C07307=1196.798,-117.716,-38.515,179.057,5.551,149.259
C07308=1196.792,-117.467,-38.525,179.060,5.552,149.258
C07309=1196.787,-117.217,-38.534,179.061,5.552,149.258
C07310=1196.782,-116.967,-38.543,179.064,5.552,149.257
C07311=1196.777,-116.718,-38.553,179.066,5.552,149.256
C07312=1196.771,-116.468,-38.562,179.068,5.553,149.256
C07313=1196.766,-116.219,-38.572,179.070,5.552,149.255
C07314=1196.761,-115.968,-38.581,179.072,5.553,149.255
C07315=1196.755,-115.718,-38.590,179.075,5.553,149.254
C07316=1196.750,-115.469,-38.600,179.077,5.553,149.253
C07317=1196.745,-115.219,-38.609,179.079,5.553,149.253
C07318=1196.739,-114.969,-38.618,179.081,5.553,149.252
C07319=1196.734,-114.719,-38.629,179.084,5.553,149.251
C07320=1196.729,-114.469,-38.637,179.086,5.554,149.251
C07321=1196.724,-114.220,-38.648,179.088,5.553,149.250
C07322=1196.719,-113.970,-38.657,179.090,5.554,149.250
C07323=1196.714,-113.721,-38.666,179.092,5.554,149.249
C07324=1196.708,-113.470,-38.676,179.095,5.554,149.248
C07325=1196.703,-113.221,-38.685,179.096,5.554,149.248
C07326=1196.697,-112.971,-38.695,179.099,5.555,149.247
C07327=1196.692,-112.721,-38.704,179.101,5.554,149.246
C07328=1196.686,-112.472,-38.714,179.103,5.555,149.246
C07329=1196.681,-112.222,-38.723,179.105,5.555,149.245
C07330=1196.675,-111.972,-38.733,179.108,5.555,149.245
C07331=1196.670,-111.722,-38.742,179.110,5.555,149.244
C07332=1196.666,-111.472,-38.752,179.112,5.555,149.243
C07333=1196.660,-111.222,-38.761,179.114,5.555,149.243
C07334=1196.655,-110.973,-38.771,179.117,5.556,149.242
C07335=1196.649,-110.723,-38.780,179.119,5.555,149.241
C07336=1196.645,-110.474,-38.790,179.121,5.556,149.241
C07337=1196.639,-110.223,-38.800,179.123,5.556,149.240
C07338=1196.634,-109.974,-38.809,179.125,5.557,149.240
C07339=1196.628,-109.724,-38.819,179.127,5.556,149.239
C07340=1196.624,-109.474,-38.829,179.130,5.557,149.238
C07341=1196.618,-109.224,-38.838,179.132,5.557,149.238
C07342=1196.613,-108.975,-38.848,179.134,5.557,149.237
C07343=1196.607,-108.725,-38.858,179.136,5.557,149.236
C07344=1196.602,-108.475,-38.867,179.139,5.557,149.236
C07345=1196.596,-108.226,-38.877,179.141,5.557,149.235
C07346=1196.591,-107.976,-38.886,179.143,5.557,149.234
C07347=1196.586,-107.726,-38.897,179.145,5.557,149.234
C07348=1196.581,-107.476,-38.906,179.148,5.558,149.233
C07349=1196.576,-107.226,-38.916,179.149,5.558,149.233
C07350=1196.570,-106.977,-38.926,179.152,5.558,149.232
C07351=1196.565,-106.727,-38.935,179.154,5.558,149.231
C07352=1196.559,-106.477,-38.945,179.156,5.559,149.231
C07353=1196.554,-106.228,-38.955,179.158,5.558,149.230
C07354=1196.549,-105.977,-38.964,179.161,5.559,149.229
C07355=1196.544,-105.728,-38.974,179.163,5.559,149.229
C07356=1196.539,-105.478,-38.984,179.165,5.559,149.228
C07357=1196.533,-105.229,-38.993,179.167,5.559,149.227
C07358=1196.528,-104.979,-39.003,179.169,5.559,149.227
C07359=1196.523,-104.729,-39.014,179.172,5.559,149.226
C07360=1196.518,-104.479,-39.023,179.174,5.559,149.225
C07361=1196.512,-104.229,-39.033,179.176,5.560,149.225
C07362=1196.507,-103.980,-39.043,179.178,5.560,149.224
C07363=1196.501,-103.730,-39.052,179.181,5.560,149.224
C07364=1196.496,-103.480,-39.063,179.183,5.560,149.223
C07365=1196.491,-103.231,-39.072,179.185,5.561,149.222
C07366=1196.486,-102.980,-39.082,179.188,5.560,149.222
C07367=1196.481,-102.731,-39.091,179.190,5.561,149.221
C07368=1196.476,-102.481,-39.102,179.192,5.561,149.220
C07369=1196.470,-102.231,-39.112,179.194,5.561,149.220
C07370=1196.465,-101.982,-39.121,179.196,5.561,149.219
C07371=1196.459,-101.710,-39.133,179.199,5.561,149.219
C07372=1196.453,-101.439,-39.143,179.201,5.562,149.218
C07373=1196.448,-101.167,-39.153,179.204,5.561,149.217
C07374=1196.442,-100.896,-39.165,179.206,5.562,149.216
C07375=1196.437,-100.647,-39.175,179.208,5.562,149.216
C07376=1196.431,-100.396,-39.184,179.210,5.562,149.215
C07377=1196.426,-100.146,-39.195,179.213,5.562,149.215
C07378=1196.421,-99.897,-39.204,179.215,5.562,149.214
C07379=1196.416,-99.647,-39.214,179.217,5.563,149.213
C07380=1196.410,-99.398,-39.225,179.220,5.563,149.213
C07381=1196.406,-99.148,-39.235,179.222,5.563,149.212
C07382=1196.400,-98.898,-39.244,179.224,5.563,149.211
C07383=1196.394,-98.648,-39.254,179.226,5.563,149.211
C07384=1196.389,-98.398,-39.265,179.229,5.563,149.210
C07385=1196.384,-98.149,-39.275,179.231,5.564,149.209
C07386=1196.379,-97.899,-39.285,179.233,5.563,149.209
C07387=1196.373,-97.650,-39.295,179.236,5.564,149.208
C07388=1196.369,-97.399,-39.304,179.237,5.564,149.208
C07389=1196.363,-97.150,-39.314,179.240,5.564,149.207
C07390=1196.357,-96.900,-39.325,179.242,5.564,149.206
C07391=1196.352,-96.650,-39.335,179.244,5.565,149.206
C07392=1196.347,-96.401,-39.345,179.246,5.564,149.205
C07393=1196.342,-96.151,-39.355,179.249,5.565,149.204
C07394=1196.336,-95.901,-39.365,179.251,5.565,149.204
C07395=1196.331,-95.651,-39.376,179.253,5.565,149.203
C07396=1196.326,-95.402,-39.386,179.256,5.565,149.202
C07397=1196.321,-95.152,-39.396,179.257,5.565,149.202
C07398=1196.316,-94.902,-39.406,179.260,5.566,149.201
C07399=1196.310,-94.652,-39.416,179.262,5.566,149.200
C07400=1196.304,-94.402,-39.426,179.265,5.566,149.200
C07401=1196.300,-94.153,-39.436,179.266,5.566,149.199
C07402=1196.294,-93.903,-39.446,179.269,5.566,149.199
C07403=1196.289,-93.653,-39.456,179.271,5.566,149.198
C07404=1196.284,-93.403,-39.467,179.273,5.567,149.197
C07405=1196.278,-93.154,-39.477,179.276,5.567,149.197
C07406=1196.273,-92.904,-39.487,179.278,5.567,149.196
C07407=1196.268,-92.654,-39.497,179.280,5.568,149.195
C07408=1196.263,-92.405,-39.508,179.282,5.567,149.195
C07409=1196.257,-92.155,-39.518,179.285,5.568,149.194
C07410=1196.252,-91.905,-39.528,179.287,5.568,149.194
C07411=1196.247,-91.655,-39.539,179.289,5.568,149.193
C07412=1196.241,-91.406,-39.549,179.291,5.568,149.192
C07413=1196.237,-91.156,-39.559,179.294,5.568,149.191
C07414=1196.231,-90.906,-39.569,179.296,5.569,149.191
C07415=1196.226,-90.656,-39.579,179.298,5.568,149.190
C07416=1196.221,-90.406,-39.590,179.301,5.569,149.189
C07417=1196.215,-90.158,-39.601,179.303,5.569,149.189
C07418=1196.210,-89.907,-39.611,179.305,5.569,149.188
C07419=1196.205,-89.658,-39.621,179.307,5.569,149.188
C07420=1196.200,-89.408,-39.631,179.310,5.569,149.187
C07421=1196.195,-89.158,-39.642,179.312,5.569,149.186
C07422=1196.189,-88.909,-39.652,179.314,5.570,149.186
C07423=1196.184,-88.659,-39.662,179.317,5.570,149.185
C07424=1196.179,-88.409,-39.673,179.319,5.570,149.184
C07425=1196.174,-88.159,-39.683,179.321,5.571,149.184
C07426=1196.168,-87.909,-39.693,179.323,5.570,149.183
C07427=1196.163,-87.660,-39.704,179.326,5.571,149.183
C07428=1196.158,-87.410,-39.715,179.328,5.571,149.182
C07429=1196.152,-87.160,-39.725,179.330,5.571,149.181
C07430=1196.147,-86.910,-39.736,179.333,5.571,149.180
C07431=1196.142,-86.661,-39.745,179.335,5.571,149.180
C07432=1196.137,-86.411,-39.756,179.337,5.572,149.179
C07433=1196.132,-86.162,-39.767,179.339,5.571,149.179
C07434=1196.126,-85.912,-39.777,179.342,5.572,149.178
C07435=1196.121,-85.662,-39.788,179.344,5.572,149.177
C07436=1196.116,-85.413,-39.798,179.346,5.572,149.177
C07437=1196.111,-85.162,-39.808,179.349,5.573,149.176
C07438=1196.106,-84.913,-39.819,179.351,5.573,149.175
C07439=1196.101,-84.663,-39.830,179.353,5.573,149.175
C07440=1196.095,-84.414,-39.840,179.355,5.573,149.174
C07441=1196.090,-84.163,-39.851,179.358,5.573,149.173
C07442=1196.084,-83.914,-39.861,179.360,5.573,149.173
C07443=1196.080,-83.664,-39.872,179.362,5.574,149.172
C07444=1196.074,-83.415,-39.882,179.365,5.574,149.171
C07445=1196.069,-83.164,-39.893,179.367,5.574,149.171
C07446=1196.063,-82.915,-39.903,179.369,5.574,149.170
C07447=1196.059,-82.665,-39.914,179.371,5.574,149.170
C07448=1196.053,-82.416,-39.925,179.374,5.575,149.169
C07449=1196.048,-82.166,-39.935,179.376,5.575,149.168
C07450=1196.043,-81.916,-39.946,179.378,5.575,149.168
C07451=1196.037,-81.667,-39.956,179.381,5.575,149.167
C07452=1196.032,-81.417,-39.967,179.383,5.575,149.166
C07453=1196.027,-81.167,-39.977,179.385,5.576,149.166
C07454=1196.022,-80.918,-39.988,179.387,5.575,149.165
C07455=1196.016,-80.668,-39.999,179.390,5.576,149.164
C07456=1196.011,-80.418,-40.009,179.392,5.577,149.164
C07457=1196.006,-80.168,-40.021,179.394,5.576,149.163
C07458=1196.000,-79.918,-40.031,179.397,5.577,149.162
C07459=1195.996,-79.669,-40.043,179.399,5.576,149.162
C07460=1195.990,-79.419,-40.053,179.401,5.577,149.161
C07461=1195.985,-79.169,-40.063,179.404,5.578,149.161
C07462=1195.980,-78.920,-40.074,179.406,5.577,149.160
C07463=1195.975,-78.670,-40.085,179.409,5.578,149.159
C07464=1195.969,-78.420,-40.095,179.410,5.578,149.159
C07465=1195.964,-78.170,-40.106,179.413,5.578,149.158
C07466=1195.959,-77.921,-40.117,179.415,5.578,149.157
C07467=1195.953,-77.671,-40.128,179.418,5.578,149.156
C07468=1195.948,-77.421,-40.139,179.420,5.579,149.156
C07469=1195.943,-77.171,-40.149,179.422,5.578,149.155
C07470=1195.938,-76.922,-40.160,179.425,5.579,149.155
C07471=1195.933,-76.672,-40.171,179.426,5.579,149.154
C07472=1195.928,-76.422,-40.182,179.429,5.579,149.153
C07473=1195.922,-76.173,-40.192,179.431,5.580,149.153
C07474=1195.917,-75.923,-40.204,179.434,5.579,149.152
C07475=1195.911,-75.652,-40.215,179.436,5.580,149.151
C07476=1195.905,-75.381,-40.227,179.439,5.580,149.151
C07477=1195.900,-75.110,-40.239,179.442,5.581,149.150
C07478=1195.894,-74.840,-40.250,179.444,5.580,149.149
C07479=1195.889,-74.590,-40.262,179.446,5.581,149.149
C07480=1195.884,-74.340,-40.273,179.448,5.581,149.148
C07481=1195.878,-74.091,-40.283,179.451,5.581,149.147
C07482=1195.874,-73.841,-40.294,179.453,5.582,149.147
C07483=1195.868,-73.592,-40.305,179.455,5.582,149.146
C07484=1195.863,-73.342,-40.316,179.458,5.582,149.145
C07485=1195.858,-73.091,-40.327,179.460,5.582,149.145
C07486=1195.852,-72.842,-40.338,179.462,5.582,149.144
C07487=1195.847,-72.592,-40.349,179.464,5.583,149.143
C07488=1195.841,-72.343,-40.360,179.467,5.583,149.143
C07489=1195.837,-72.093,-40.371,179.469,5.583,149.142
C07490=1195.832,-71.843,-40.382,179.472,5.583,149.141
C07491=1195.826,-71.594,-40.393,179.473,5.583,149.141
C07492=1195.821,-71.344,-40.404,179.476,5.584,149.140
C07493=1195.815,-71.095,-40.415,179.478,5.583,149.139
C07494=1195.810,-70.844,-40.426,179.481,5.584,149.139
C07495=1195.806,-70.595,-40.437,179.483,5.585,149.138
C07496=1195.800,-70.346,-40.448,179.485,5.584,149.138
C07497=1195.795,-70.095,-40.459,179.488,5.585,149.137
C07498=1195.790,-69.846,-40.470,179.491,5.585,149.136
C07499=1195.785,-69.597,-40.481,179.492,5.585,149.136
C07500=1195.779,-69.346,-40.492,179.495,5.586,149.135
C07501=1195.774,-69.097,-40.504,179.497,5.585,149.134
C07502=1195.769,-68.848,-40.515,179.500,5.586,149.134
C07503=1195.763,-68.597,-40.526,179.502,5.586,149.133
C07504=1195.758,-68.347,-40.537,179.504,5.586,149.132
C07505=1195.753,-68.099,-40.548,179.506,5.587,149.132
C07506=1195.747,-67.848,-40.559,179.509,5.587,149.131
C07507=1195.743,-67.598,-40.570,179.511,5.587,149.130
C07508=1195.737,-67.349,-40.581,179.513,5.587,149.130
C07509=1195.732,-67.099,-40.592,179.515,5.587,149.129
C07510=1195.727,-66.849,-40.604,179.518,5.587,149.128
C07511=1195.722,-66.600,-40.615,179.521,5.588,149.128
C07512=1195.716,-66.350,-40.627,179.522,5.588,149.127
C07513=1195.711,-66.100,-40.637,179.525,5.588,149.126
C07514=1195.707,-65.851,-40.648,179.528,5.589,149.126
C07515=1195.701,-65.601,-40.660,179.530,5.588,149.125
C07516=1195.696,-65.352,-40.671,179.532,5.589,149.125
C07517=1195.691,-65.101,-40.682,179.535,5.590,149.124
C07518=1195.685,-64.851,-40.694,179.537,5.589,149.123
C07519=1195.680,-64.603,-40.705,179.539,5.590,149.122
C07520=1195.675,-64.353,-40.717,179.541,5.590,149.122
C07521=1195.670,-64.102,-40.727,179.544,5.590,149.121
C07522=1195.664,-63.853,-40.738,179.546,5.591,149.121
C07523=1195.659,-63.604,-40.750,179.548,5.590,149.120
C07524=1195.654,-63.354,-40.761,179.551,5.591,149.119
C07525=1195.649,-63.104,-40.773,179.553,5.592,149.119
C07526=1195.644,-62.855,-40.784,179.555,5.591,149.118
C07527=1195.639,-62.605,-40.795,179.558,5.592,149.117
C07528=1195.633,-62.355,-40.806,179.561,5.592,149.117
C07529=1195.628,-62.105,-40.818,179.562,5.592,149.116
C07530=1195.623,-61.855,-40.830,179.565,5.592,149.115
C07531=1195.618,-61.606,-40.841,179.568,5.593,149.115
C07532=1195.612,-61.356,-40.852,179.570,5.593,149.114
C07533=1195.608,-61.107,-40.864,179.572,5.593,149.113
C07534=1195.602,-60.856,-40.875,179.575,5.594,149.113
C07535=1195.597,-60.607,-40.886,179.577,5.593,149.112
C07536=1195.591,-60.357,-40.898,179.579,5.594,149.111
C07537=1195.586,-60.108,-40.909,179.582,5.594,149.111
C07538=1195.582,-59.858,-40.920,179.584,5.594,149.110
C07539=1195.576,-59.608,-40.932,179.586,5.595,149.109
C07540=1195.571,-59.359,-40.943,179.588,5.594,149.109
C07541=1195.566,-59.109,-40.955,179.591,5.595,149.108
C07542=1195.561,-58.860,-40.966,179.593,5.596,149.108
C07543=1195.556,-58.610,-40.978,179.595,5.595,149.107
C07544=1195.551,-58.360,-40.989,179.598,5.596,149.106
C07545=1195.545,-58.110,-41.001,179.601,5.596,149.105
C07546=1195.540,-57.861,-41.012,179.603,5.596,149.105
C07547=1195.535,-57.611,-41.024,179.605,5.597,149.104
C07548=1195.529,-57.361,-41.036,179.608,5.597,149.104
C07549=1195.525,-57.112,-41.047,179.610,5.597,149.103
C07550=1195.519,-56.862,-41.059,179.612,5.597,149.102
C07551=1195.514,-56.612,-41.070,179.614,5.598,149.102
C07552=1195.508,-56.363,-41.082,179.617,5.598,149.101
C07553=1195.504,-56.113,-41.093,179.619,5.598,149.100
C07554=1195.498,-55.863,-41.105,179.622,5.598,149.100
C07555=1195.494,-55.614,-41.116,179.624,5.598,149.099
C07556=1195.488,-55.364,-41.128,179.626,5.599,149.098
C07557=1195.483,-55.114,-41.140,179.629,5.599,149.098
C07558=1195.478,-54.864,-41.152,179.631,5.599,149.097
C07559=1195.472,-54.615,-41.163,179.634,5.599,149.096
C07560=1195.467,-54.365,-41.174,179.636,5.600,149.096
C07561=1195.462,-54.116,-41.186,179.638,5.601,149.095
C07562=1195.457,-53.866,-41.198,179.640,5.600,149.094
C07563=1195.452,-53.616,-41.209,179.643,5.601,149.094
C07564=1195.447,-53.367,-41.222,179.646,5.601,149.093
C07565=1195.442,-53.117,-41.233,179.647,5.601,149.093
C07566=1195.437,-52.867,-41.245,179.650,5.602,149.092
C07567=1195.431,-52.617,-41.257,179.653,5.602,149.091
C07568=1195.426,-52.368,-41.268,179.655,5.602,149.090
C07569=1195.420,-52.118,-41.280,179.657,5.602,149.090
C07570=1195.416,-51.869,-41.291,179.660,5.603,149.089
C07571=1195.410,-51.619,-41.303,179.662,5.603,149.089
C07572=1195.405,-51.369,-41.316,179.664,5.603,149.088
C07573=1195.400,-51.120,-41.327,179.667,5.604,149.087
C07574=1195.395,-50.870,-41.339,179.669,5.604,149.087
C07575=1195.390,-50.620,-41.351,179.671,5.604,149.086
C07576=1195.385,-50.370,-41.362,179.674,5.604,149.085
C07577=1195.380,-50.121,-41.375,179.677,5.605,149.085
C07578=1195.374,-49.871,-41.386,179.679,5.605,149.084
C07579=1195.368,-49.601,-41.399,179.681,5.605,149.083
C07580=1195.363,-49.331,-41.412,179.684,5.605,149.082
C07581=1195.358,-49.061,-41.425,179.687,5.606,149.082
C07582=1195.352,-48.791,-41.438,179.689,5.606,149.081
C07583=1195.346,-48.541,-41.450,179.691,5.606,149.081
C07584=1195.341,-48.291,-41.461,179.694,5.607,149.080
C07585=1195.336,-48.042,-41.473,179.696,5.607,149.079
C07586=1195.331,-47.792,-41.485,179.698,5.607,149.078
C07587=1195.326,-47.542,-41.497,179.701,5.607,149.078
C07588=1195.320,-47.292,-41.509,179.703,5.608,149.077
C07589=1195.316,-47.043,-41.520,179.705,5.608,149.077
C07590=1195.311,-46.793,-41.533,179.708,5.608,149.076
C07591=1195.305,-46.543,-41.545,179.711,5.609,149.075
C07592=1195.300,-46.294,-41.557,179.713,5.609,149.074
C07593=1195.295,-46.045,-41.569,179.715,5.609,149.074
C07594=1195.290,-45.795,-41.581,179.718,5.610,149.073
C07595=1195.284,-45.545,-41.592,179.720,5.610,149.073
C07596=1195.279,-45.295,-41.605,179.722,5.610,149.072
C07597=1195.274,-45.045,-41.617,179.725,5.610,149.071
C07598=1195.269,-44.796,-41.628,179.727,5.611,149.071
C07599=1195.264,-44.546,-41.641,179.730,5.611,149.070
C07600=1195.259,-44.296,-41.653,179.732,5.611,149.069
C07601=1195.253,-44.047,-41.665,179.735,5.612,149.069
C07602=1195.248,-43.797,-41.677,179.737,5.612,149.068
C07603=1195.243,-43.548,-41.689,179.739,5.612,149.067
C07604=1195.238,-43.298,-41.701,179.742,5.612,149.067
C07605=1195.233,-43.048,-41.713,179.744,5.613,149.066
C07606=1195.227,-42.798,-41.725,179.747,5.613,149.065
C07607=1195.222,-42.549,-41.737,179.749,5.613,149.065
C07608=1195.217,-42.299,-41.749,179.751,5.614,149.064
C07609=1195.212,-42.050,-41.761,179.754,5.614,149.063
C07610=1195.207,-41.800,-41.773,179.756,5.614,149.063
C07611=1195.202,-41.551,-41.786,179.759,5.614,149.062
C07612=1195.196,-41.301,-41.798,179.761,5.615,149.062
C07613=1195.191,-41.052,-41.810,179.763,5.616,149.061
C07614=1195.186,-40.802,-41.822,179.765,5.615,149.060
C07615=1195.181,-40.552,-41.835,179.768,5.616,149.059
C07616=1195.176,-40.302,-41.847,179.771,5.616,149.059
C07617=1195.171,-40.052,-41.860,179.773,5.617,149.058
C07618=1195.166,-39.803,-41.871,179.775,5.617,149.058
C07619=1195.161,-39.554,-41.884,179.778,5.617,149.057
C07620=1195.156,-39.304,-41.895,179.780,5.618,149.056
C07621=1195.150,-39.054,-41.908,179.783,5.618,149.056
C07622=1195.145,-38.804,-41.920,179.785,5.618,149.055
C07623=1195.140,-38.555,-41.933,179.787,5.619,149.054
C07624=1195.134,-38.305,-41.944,179.790,5.619,149.054
C07625=1195.129,-38.056,-41.957,179.792,5.619,149.053
C07626=1195.124,-37.806,-41.969,179.795,5.619,149.052
C07627=1195.119,-37.556,-41.982,179.797,5.620,149.052
C07628=1195.114,-37.306,-41.994,179.800,5.620,149.051
C07629=1195.109,-37.057,-42.006,179.802,5.620,149.050
C07630=1195.104,-36.807,-42.019,179.804,5.621,149.050
C07631=1195.098,-36.557,-42.031,179.807,5.621,149.049
C07632=1195.093,-36.308,-42.043,179.809,5.622,149.048
C07633=1195.088,-36.059,-42.056,179.811,5.621,149.048
C07634=1195.083,-35.809,-42.068,179.814,5.622,149.047
C07635=1195.078,-35.559,-42.081,179.816,5.622,149.046
C07636=1195.073,-35.309,-42.093,179.819,5.623,149.046
C07637=1195.068,-35.059,-42.105,179.821,5.623,149.045
C07638=1195.062,-34.810,-42.118,179.823,5.623,149.045
C07639=1195.057,-34.560,-42.130,179.826,5.624,149.044
C07640=1195.052,-34.311,-42.142,179.829,5.624,149.043
C07641=1195.047,-34.062,-42.155,179.831,5.624,149.042
C07642=1195.042,-33.812,-42.168,179.833,5.625,149.042
C07643=1195.037,-33.562,-42.180,179.836,5.625,149.041
C07644=1195.032,-33.312,-42.193,179.838,5.626,149.041
C07645=1195.027,-33.063,-42.205,179.841,5.626,149.040
C07646=1195.021,-32.813,-42.217,179.843,5.626,149.039
C07647=1195.016,-32.564,-42.230,179.845,5.627,149.039
C07648=1195.011,-32.314,-42.243,179.848,5.627,149.038
C07649=1195.006,-32.064,-42.255,179.851,5.628,149.037
C07650=1195.001,-31.814,-42.267,179.853,5.627,149.037
C07651=1194.996,-31.565,-42.280,179.855,5.628,149.036
C07652=1194.990,-31.315,-42.293,179.857,5.628,149.035
C07653=1194.985,-31.065,-42.306,179.860,5.629,149.035
C07654=1194.980,-30.816,-42.318,179.862,5.629,149.034
C07655=1194.975,-30.566,-42.330,179.865,5.629,149.033
C07656=1194.970,-30.317,-42.343,179.868,5.630,149.033
C07657=1194.965,-30.068,-42.356,179.870,5.630,149.032
C07658=1194.960,-29.818,-42.369,179.872,5.630,149.031
C07659=1194.955,-29.568,-42.380,179.874,5.630,149.031
C07660=1194.950,-29.318,-42.393,179.877,5.631,149.030
C07661=1194.944,-29.069,-42.406,179.880,5.631,149.029
C07662=1194.939,-28.819,-42.419,179.882,5.632,149.029
C07663=1194.934,-28.569,-42.432,179.884,5.632,149.028
C07664=1194.929,-28.320,-42.444,179.887,5.632,149.028
C07665=1194.923,-28.070,-42.456,179.889,5.633,149.027
C07666=1194.919,-27.820,-42.469,179.892,5.633,149.026
C07667=1194.913,-27.570,-42.482,179.894,5.633,149.025
C07668=1194.908,-27.321,-42.495,179.896,5.634,149.025
C07669=1194.903,-27.072,-42.508,179.899,5.634,149.024
C07670=1194.898,-26.822,-42.521,179.902,5.635,149.024
C07671=1194.893,-26.572,-42.533,179.904,5.635,149.023
C07672=1194.888,-26.323,-42.546,179.906,5.635,149.022
C07673=1194.882,-26.074,-42.559,179.908,5.636,149.022
C07674=1194.878,-25.823,-42.572,179.911,5.636,149.021
C07675=1194.873,-25.574,-42.585,179.914,5.637,149.020
C07676=1194.867,-25.324,-42.596,179.916,5.637,149.020
C07677=1194.862,-25.074,-42.610,179.919,5.637,149.019
C07678=1194.857,-24.825,-42.623,179.921,5.638,149.018
C07679=1194.852,-24.575,-42.635,179.923,5.638,149.018
C07680=1194.847,-24.325,-42.648,179.926,5.638,149.017
C07681=1194.842,-24.076,-42.661,179.929,5.639,149.016
C07682=1194.836,-23.826,-42.674,179.931,5.639,149.016
C07683=1194.831,-23.557,-42.688,179.933,5.639,149.015
C07684=1194.825,-23.287,-42.702,179.936,5.640,149.014
C07685=1194.820,-23.018,-42.716,179.939,5.640,149.014
C07686=1194.814,-22.748,-42.730,179.941,5.640,149.013
C07687=1194.809,-22.499,-42.743,179.944,5.641,149.012
C07688=1194.805,-22.249,-42.756,179.946,5.642,149.012
C07689=1194.799,-21.999,-42.769,179.949,5.642,149.011
C07690=1194.794,-21.750,-42.782,179.951,5.642,149.010
C07691=1194.789,-21.500,-42.795,179.954,5.642,149.010
C07692=1194.784,-21.250,-42.807,179.956,5.643,149.009
C07693=1194.778,-21.001,-42.820,179.958,5.644,149.008
C07694=1194.774,-20.751,-42.833,179.961,5.644,149.008
C07695=1194.769,-20.502,-42.846,179.963,5.644,149.007
C07696=1194.763,-20.252,-42.859,179.966,5.644,149.006
C07697=1194.758,-20.002,-42.872,179.968,5.645,149.006
C07698=1194.753,-19.753,-42.885,179.971,5.646,149.005
C07699=1194.747,-19.504,-42.899,179.973,5.646,149.005
C07700=1194.743,-19.254,-42.912,179.976,5.647,149.004
C07701=1194.737,-19.004,-42.925,179.978,5.646,149.003
C07702=1194.732,-18.755,-42.937,179.980,5.647,149.003
C07703=1194.727,-18.505,-42.950,179.983,5.648,149.002
C07704=1194.722,-18.255,-42.964,179.986,5.648,149.001
C07705=1194.717,-18.006,-42.977,179.988,5.648,149.001
C07706=1194.712,-17.756,-42.990,179.990,5.648,149.000
C07707=1194.706,-17.507,-43.003,179.992,5.649,148.999
C07708=1194.702,-17.257,-43.016,179.995,5.649,148.999
C07709=1194.696,-17.007,-43.029,179.998,5.650,148.998
C07710=1194.692,-16.758,-43.043,-180.000,5.650,148.997
C07711=1194.686,-16.508,-43.056,-179.997,5.651,148.997
C07712=1194.681,-16.258,-43.069,-179.995,5.651,148.996
C07713=1194.676,-16.009,-43.082,-179.993,5.651,148.995
C07714=1194.671,-15.760,-43.095,-179.990,5.652,148.995
C07715=1194.666,-15.510,-43.108,-179.987,5.652,148.994
C07716=1194.660,-15.260,-43.122,-179.985,5.653,148.993
C07717=1194.656,-15.010,-43.135,-179.982,5.654,148.993
C07718=1194.650,-14.761,-43.149,-179.980,5.653,148.992
C07719=1194.646,-14.511,-43.162,-179.978,5.654,148.992
C07720=1194.641,-14.262,-43.174,-179.975,5.654,148.991
C07721=1194.635,-14.013,-43.188,-179.972,5.655,148.990
C07722=1194.631,-13.763,-43.201,-179.970,5.656,148.990
C07723=1194.625,-13.513,-43.214,-179.968,5.656,148.989
C07724=1194.620,-13.263,-43.227,-179.965,5.657,148.988
C07725=1194.615,-13.014,-43.241,-179.963,5.656,148.988
C07726=1194.610,-12.764,-43.254,-179.960,5.657,148.987
C07727=1194.604,-12.514,-43.267,-179.958,5.658,148.986
C07728=1194.600,-12.265,-43.281,-179.955,5.658,148.986
C07729=1194.594,-12.015,-43.294,-179.953,5.658,148.985
C07730=1194.590,-11.766,-43.308,-179.950,5.659,148.984
C07731=1194.584,-11.516,-43.321,-179.948,5.659,148.984
C07732=1194.580,-11.266,-43.334,-179.946,5.659,148.983
C07733=1194.574,-11.017,-43.348,-179.943,5.660,148.983
C07734=1194.569,-10.767,-43.361,-179.941,5.660,148.982
C07735=1194.564,-10.518,-43.375,-179.938,5.661,148.981
C07736=1194.559,-10.268,-43.388,-179.935,5.661,148.980
C07737=1194.554,-10.018,-43.401,-179.933,5.662,148.980
C07738=1194.549,-9.769,-43.415,-179.931,5.662,148.979
C07739=1194.543,-9.519,-43.428,-179.928,5.662,148.979
C07740=1194.538,-9.270,-43.442,-179.926,5.663,148.978
C07741=1194.533,-9.020,-43.455,-179.923,5.663,148.977
C07742=1194.528,-8.771,-43.469,-179.921,5.664,148.977
C07743=1194.523,-8.521,-43.482,-179.918,5.665,148.976
C07744=1194.518,-8.272,-43.496,-179.916,5.665,148.975
C07745=1194.513,-8.021,-43.509,-179.913,5.666,148.975
C07746=1194.508,-7.773,-43.523,-179.911,5.665,148.974
C07747=1194.503,-7.522,-43.536,-179.909,5.666,148.974
C07748=1194.497,-7.273,-43.550,-179.906,5.667,148.973
C07749=1194.493,-7.023,-43.563,-179.903,5.667,148.972
C07750=1194.487,-6.774,-43.577,-179.901,5.668,148.971
C07751=1194.482,-6.524,-43.591,-179.898,5.668,148.971
C07752=1194.477,-6.275,-43.604,-179.896,5.669,148.970
C07753=1194.472,-6.025,-43.617,-179.893,5.669,148.970
C07754=1194.467,-5.775,-43.632,-179.891,5.669,148.969
C07755=1194.462,-5.526,-43.644,-179.888,5.670,148.968
C07756=1194.457,-5.276,-43.659,-179.886,5.670,148.968
C07757=1194.451,-5.027,-43.673,-179.884,5.671,148.967
C07758=1194.447,-4.777,-43.686,-179.881,5.671,148.966
C07759=1194.442,-4.527,-43.700,-179.878,5.672,148.966
C07760=1194.436,-4.278,-43.713,-179.876,5.672,148.965
C07761=1194.432,-4.028,-43.727,-179.874,5.673,148.965
C07762=1194.426,-3.779,-43.741,-179.871,5.673,148.964
C07763=1194.421,-3.529,-43.754,-179.869,5.673,148.963
C07764=1194.417,-3.280,-43.768,-179.866,5.674,148.962
C07765=1194.411,-3.031,-43.782,-179.863,5.674,148.962
C07766=1194.406,-2.780,-43.795,-179.861,5.675,148.961
C07767=1194.400,-2.531,-43.809,-179.859,5.676,148.961
C07768=1194.396,-2.282,-43.823,-179.856,5.676,148.960
C07769=1194.391,-2.032,-43.836,-179.853,5.677,148.959
C07770=1194.385,-1.783,-43.850,-179.851,5.677,148.959
C07771=1194.380,-1.533,-43.865,-179.849,5.678,148.958
C07772=1194.376,-1.283,-43.878,-179.846,5.678,148.957
C07773=1194.370,-1.034,-43.892,-179.844,5.678,148.957
C07774=1194.365,-0.784,-43.906,-179.841,5.679,148.956
C07775=1194.360,-0.534,-43.920,-179.838,5.679,148.955
C07776=1194.355,-0.285,-43.933,-179.836,5.680,148.955
C07777=1194.350,-0.035,-43.947,-179.834,5.680,148.954
C07778=1194.345,0.214,-43.961,-179.831,5.681,148.954
C07779=1194.340,0.463,-43.975,-179.828,5.681,148.953
C07780=1194.335,0.714,-43.989,-179.826,5.682,148.952
C07781=1194.330,0.963,-44.002,-179.824,5.683,148.952
C07782=1194.325,1.212,-44.016,-179.821,5.682,148.951
C07783=1194.320,1.462,-44.031,-179.819,5.683,148.950
C07784=1194.315,1.711,-44.045,-179.816,5.683,148.950
C07785=1194.309,1.961,-44.058,-179.814,5.684,148.949
C07786=1194.304,2.211,-44.072,-179.811,5.685,148.948
C07787=1194.299,2.480,-44.087,-179.809,5.685,148.948
C07788=1194.294,2.749,-44.103,-179.806,5.686,148.947
C07789=1194.288,3.017,-44.117,-179.803,5.686,148.946
C07790=1194.283,3.287,-44.132,-179.801,5.687,148.946
C07791=1194.278,3.537,-44.146,-179.798,5.687,148.945
C07792=1194.273,3.786,-44.161,-179.795,5.688,148.944
C07793=1194.267,4.035,-44.175,-179.793,5.688,148.944
C07794=1194.262,4.285,-44.189,-179.791,5.689,148.943
C07795=1194.257,4.535,-44.202,-179.788,5.690,148.943
C07796=1194.252,4.785,-44.217,-179.785,5.690,148.942
C07797=1194.247,5.034,-44.231,-179.783,5.690,148.941
C07798=1194.242,5.284,-44.245,-179.780,5.691,148.941
C07799=1194.237,5.533,-44.258,-179.778,5.692,148.940
C07800=1194.233,5.783,-44.273,-179.775,5.692,148.939
C07801=1194.227,6.032,-44.287,-179.773,5.693,148.939
C07802=1194.222,6.282,-44.301,-179.770,5.693,148.938
C07803=1194.217,6.531,-44.315,-179.768,5.694,148.937
C07804=1194.212,6.781,-44.330,-179.766,5.694,148.937
C07805=1194.207,7.030,-44.343,-179.763,5.694,148.936
C07806=1194.202,7.280,-44.358,-179.760,5.695,148.935
C07807=1194.197,7.529,-44.372,-179.758,5.696,148.935
C07808=1194.192,7.779,-44.386,-179.756,5.696,148.934
C07809=1194.186,8.028,-44.400,-179.753,5.697,148.934
C07810=1194.181,8.278,-44.414,-179.750,5.697,148.933
C07811=1194.176,8.528,-44.429,-179.748,5.698,148.932
C07812=1194.171,8.777,-44.443,-179.745,5.699,148.932
C07813=1194.166,9.027,-44.457,-179.743,5.699,148.931
C07814=1194.161,9.276,-44.471,-179.740,5.700,148.930
C07815=1194.156,9.526,-44.485,-179.737,5.700,148.930
C07816=1194.151,9.775,-44.500,-179.735,5.701,148.929
C07817=1194.146,10.025,-44.514,-179.733,5.701,148.929
C07818=1194.141,10.275,-44.528,-179.730,5.702,148.928
C07819=1194.136,10.525,-44.543,-179.727,5.702,148.927
C07820=1194.130,10.774,-44.556,-179.725,5.703,148.927
C07821=1194.126,11.023,-44.571,-179.723,5.704,148.926
C07822=1194.121,11.272,-44.586,-179.720,5.704,148.925
C07823=1194.116,11.522,-44.600,-179.717,5.705,148.925
C07824=1194.111,11.772,-44.614,-179.715,5.705,148.924
C07825=1194.106,12.021,-44.629,-179.713,5.705,148.924
C07826=1194.100,12.270,-44.642,-179.710,5.706,148.923
C07827=1194.095,12.520,-44.657,-179.708,5.706,148.922
C07828=1194.090,12.770,-44.672,-179.705,5.707,148.921
C07829=1194.085,13.019,-44.687,-179.703,5.708,148.921
C07830=1194.080,13.269,-44.701,-179.700,5.708,148.920
C07831=1194.075,13.519,-44.715,-179.698,5.709,148.920
C07832=1194.070,13.768,-44.729,-179.695,5.709,148.919
C07833=1194.065,14.017,-44.743,-179.693,5.710,148.919
C07834=1194.060,14.267,-44.758,-179.690,5.710,148.918
C07835=1194.055,14.516,-44.773,-179.687,5.711,148.917
C07836=1194.050,14.766,-44.787,-179.685,5.711,148.916
C07837=1194.044,15.016,-44.802,-179.682,5.712,148.916
C07838=1194.040,15.265,-44.817,-179.680,5.713,148.915
C07839=1194.035,15.515,-44.831,-179.677,5.713,148.915
C07840=1194.030,15.765,-44.845,-179.675,5.714,148.914
C07841=1194.025,16.014,-44.860,-179.672,5.714,148.913
C07842=1194.020,16.263,-44.875,-179.670,5.715,148.913
C07843=1194.015,16.512,-44.889,-179.667,5.716,148.912
C07844=1194.009,16.762,-44.903,-179.665,5.716,148.911
C07845=1194.004,17.011,-44.918,-179.662,5.717,148.911
C07846=1193.999,17.261,-44.933,-179.660,5.718,148.910
C07847=1193.994,17.511,-44.947,-179.657,5.718,148.910
C07848=1193.990,17.760,-44.962,-179.654,5.719,148.909
C07849=1193.984,18.010,-44.977,-179.652,5.719,148.908
C07850=1193.979,18.260,-44.991,-179.650,5.720,148.908
C07851=1193.975,18.509,-45.006,-179.647,5.720,148.907
C07852=1193.970,18.758,-45.020,-179.644,5.721,148.906
C07853=1193.965,19.008,-45.035,-179.642,5.721,148.906
C07854=1193.959,19.258,-45.050,-179.640,5.722,148.905
C07855=1193.954,19.507,-45.065,-179.637,5.723,148.905
C07856=1193.950,19.756,-45.079,-179.634,5.723,148.904
C07857=1193.945,20.006,-45.094,-179.632,5.724,148.903
C07858=1193.939,20.256,-45.109,-179.629,5.725,148.903
C07859=1193.934,20.505,-45.124,-179.627,5.725,148.902
C07860=1193.929,20.755,-45.138,-179.624,5.726,148.901
C07861=1193.924,21.004,-45.153,-179.622,5.726,148.901
C07862=1193.919,21.254,-45.168,-179.619,5.727,148.900
C07863=1193.914,21.503,-45.183,-179.617,5.728,148.900
C07864=1193.909,21.753,-45.197,-179.614,5.728,148.899
C07865=1193.904,22.003,-45.212,-179.611,5.729,148.898
C07866=1193.899,22.252,-45.227,-179.609,5.729,148.898
C07867=1193.894,22.502,-45.241,-179.607,5.730,148.897
C07868=1193.889,22.751,-45.257,-179.604,5.730,148.896
C07869=1193.884,23.001,-45.271,-179.601,5.731,148.896
C07870=1193.879,23.250,-45.286,-179.599,5.732,148.895
C07871=1193.874,23.499,-45.302,-179.597,5.732,148.895
C07872=1193.869,23.749,-45.316,-179.594,5.733,148.894
C07873=1193.864,23.998,-45.331,-179.591,5.733,148.893
C07874=1193.858,24.248,-45.346,-179.589,5.734,148.893
C07875=1193.854,24.497,-45.361,-179.586,5.735,148.892
C07876=1193.849,24.747,-45.375,-179.584,5.735,148.892
C07877=1193.843,24.996,-45.391,-179.581,5.736,148.891
C07878=1193.839,25.246,-45.405,-179.579,5.737,148.890
C07879=1193.834,25.495,-45.420,-179.576,5.737,148.890
C07880=1193.828,25.745,-45.435,-179.574,5.738,148.889
C07881=1193.824,25.994,-45.450,-179.571,5.738,148.888
C07882=1193.818,26.244,-45.465,-179.568,5.740,148.888
C07883=1193.813,26.493,-45.480,-179.566,5.740,148.887
C07884=1193.809,26.742,-45.495,-179.563,5.741,148.887
C07885=1193.803,26.992,-45.510,-179.560,5.741,148.886
C07886=1193.799,27.242,-45.525,-179.558,5.742,148.885
C07887=1193.793,27.492,-45.540,-179.556,5.743,148.885
C07888=1193.789,27.741,-45.555,-179.553,5.743,148.884
C07889=1193.783,27.991,-45.570,-179.550,5.744,148.883
C07890=1193.778,28.240,-45.585,-179.548,5.745,148.883
C07891=1193.773,28.509,-45.602,-179.545,5.745,148.882
C07892=1193.768,28.777,-45.618,-179.543,5.746,148.882
C07893=1193.762,29.046,-45.634,-179.540,5.746,148.881
C07894=1193.757,29.315,-45.650,-179.537,5.747,148.880
C07895=1193.751,29.564,-45.666,-179.534,5.748,148.880
C07896=1193.747,29.813,-45.681,-179.532,5.748,148.879
C07897=1193.741,30.063,-45.696,-179.529,5.749,148.878
C07898=1193.736,30.313,-45.710,-179.527,5.750,148.878
C07899=1193.732,30.563,-45.726,-179.524,5.750,148.877
C07900=1193.727,30.812,-45.741,-179.522,5.751,148.877
C07901=1193.722,31.061,-45.757,-179.519,5.752,148.876
C07902=1193.717,31.311,-45.771,-179.517,5.752,148.875
C07903=1193.711,31.560,-45.787,-179.514,5.753,148.875
C07904=1193.707,31.809,-45.802,-179.512,5.754,148.874
C07905=1193.701,32.059,-45.817,-179.509,5.754,148.873
C07906=1193.697,32.309,-45.833,-179.507,5.755,148.873
C07907=1193.692,32.558,-45.848,-179.504,5.755,148.872
C07908=1193.687,32.808,-45.863,-179.501,5.757,148.872
C07909=1193.681,33.057,-45.878,-179.499,5.757,148.871
C07910=1193.676,33.307,-45.894,-179.496,5.758,148.870
C07911=1193.672,33.556,-45.909,-179.494,5.759,148.870
C07912=1193.667,33.806,-45.925,-179.491,5.759,148.869
C07913=1193.662,34.055,-45.940,-179.489,5.760,148.868
C07914=1193.657,34.304,-45.955,-179.486,5.760,148.868
C07915=1193.651,34.554,-45.971,-179.484,5.761,148.867
C07916=1193.646,34.803,-45.985,-179.481,5.762,148.867
C07917=1193.641,35.053,-46.001,-179.478,5.762,148.866
C07918=1193.637,35.303,-46.016,-179.476,5.763,148.866
C07919=1193.631,35.552,-46.032,-179.474,5.764,148.865
C07920=1193.626,35.801,-46.047,-179.470,5.765,148.864
C07921=1193.622,36.051,-46.063,-179.468,5.765,148.864
C07922=1193.617,36.301,-46.078,-179.466,5.766,148.863
C07923=1193.611,36.550,-46.094,-179.463,5.767,148.862
C07924=1193.607,36.799,-46.109,-179.460,5.767,148.862
C07925=1193.601,37.048,-46.124,-179.458,5.768,148.861
C07926=1193.596,37.299,-46.140,-179.456,5.769,148.861
C07927=1193.592,37.548,-46.155,-179.453,5.769,148.860
C07928=1193.586,37.797,-46.171,-179.450,5.770,148.859
C07929=1193.581,38.046,-46.187,-179.448,5.771,148.859
C07930=1193.577,38.296,-46.202,-179.445,5.771,148.858
C07931=1193.571,38.546,-46.218,-179.442,5.773,148.857
C07932=1193.566,38.795,-46.233,-179.440,5.773,148.857
C07933=1193.561,39.044,-46.248,-179.437,5.774,148.856
C07934=1193.557,39.294,-46.264,-179.435,5.774,148.856
C07935=1193.551,39.544,-46.280,-179.432,5.775,148.855
C07936=1193.546,39.793,-46.295,-179.430,5.776,148.855
C07937=1193.542,40.043,-46.311,-179.427,5.776,148.854
C07938=1193.537,40.292,-46.327,-179.425,5.777,148.853
C07939=1193.531,40.541,-46.343,-179.423,5.778,148.853
C07940=1193.526,40.790,-46.358,-179.419,5.779,148.852
C07941=1193.522,41.040,-46.373,-179.417,5.780,148.851
C07942=1193.517,41.290,-46.389,-179.414,5.780,148.851
C07943=1193.511,41.539,-46.405,-179.412,5.781,148.850
C07944=1193.506,41.789,-46.421,-179.409,5.782,148.850
C07945=1193.502,42.038,-46.436,-179.407,5.782,148.849
C07946=1193.497,42.287,-46.452,-179.405,5.783,148.849
C07947=1193.492,42.537,-46.468,-179.402,5.783,148.848
C07948=1193.486,42.786,-46.483,-179.399,5.784,148.847
C07949=1193.481,43.036,-46.499,-179.396,5.786,148.847
C07950=1193.477,43.286,-46.514,-179.394,5.786,148.846
C07951=1193.472,43.534,-46.531,-179.391,5.787,148.845
C07952=1193.467,43.784,-46.546,-179.389,5.788,148.845
C07953=1193.462,44.034,-46.562,-179.386,5.788,148.844
C07954=1193.456,44.283,-46.578,-179.384,5.789,148.844
C07955=1193.451,44.532,-46.594,-179.381,5.789,148.843
C07956=1193.447,44.782,-46.609,-179.378,5.791,148.843
C07957=1193.442,45.031,-46.625,-179.376,5.791,148.842
C07958=1193.436,45.281,-46.641,-179.373,5.792,148.841
C07959=1193.432,45.530,-46.657,-179.371,5.793,148.841
C07960=1193.427,45.780,-46.673,-179.368,5.793,148.840
C07961=1193.422,46.030,-46.689,-179.366,5.794,148.839
C07962=1193.417,46.279,-46.705,-179.364,5.795,148.839
C07963=1193.411,46.528,-46.721,-179.361,5.795,148.838
C07964=1193.407,46.778,-46.736,-179.358,5.797,148.838
C07965=1193.402,47.026,-46.752,-179.356,5.798,148.837
C07966=1193.397,47.277,-46.768,-179.353,5.798,148.836
C07967=1193.392,47.526,-46.784,-179.350,5.799,148.836
C07968=1193.387,47.775,-46.800,-179.348,5.799,148.835
C07969=1193.382,48.025,-46.816,-179.345,5.800,148.835
C07970=1193.377,48.274,-46.832,-179.342,5.801,148.834
C07971=1193.372,48.524,-46.848,-179.340,5.802,148.833
C07972=1193.367,48.773,-46.864,-179.337,5.803,148.833
C07973=1193.362,49.023,-46.881,-179.335,5.803,148.832
C07974=1193.357,49.272,-46.896,-179.332,5.804,148.832
C07975=1193.352,49.521,-46.912,-179.330,5.805,148.831
C07976=1193.347,49.771,-46.929,-179.327,5.806,148.830
C07977=1193.342,50.020,-46.944,-179.324,5.807,148.830
C07978=1193.337,50.270,-46.961,-179.322,5.807,148.829
C07979=1193.332,50.519,-46.976,-179.319,5.808,148.829
C07980=1193.327,50.769,-46.993,-179.317,5.808,148.828
C07981=1193.322,51.018,-47.009,-179.315,5.809,148.828
C07982=1193.318,51.268,-47.025,-179.311,5.811,148.827
C07983=1193.312,51.517,-47.041,-179.309,5.811,148.826
C07984=1193.308,51.766,-47.058,-179.307,5.812,148.826
C07985=1193.302,52.016,-47.073,-179.304,5.813,148.825
C07986=1193.298,52.265,-47.090,-179.301,5.813,148.824
C07987=1193.292,52.515,-47.105,-179.299,5.814,148.824
C07988=1193.288,52.764,-47.122,-179.296,5.815,148.823
C07989=1193.283,53.014,-47.138,-179.293,5.816,148.823
C07990=1193.278,53.263,-47.154,-179.291,5.817,148.822
C07991=1193.273,53.513,-47.170,-179.289,5.817,148.822
C07992=1193.268,53.762,-47.187,-179.286,5.818,148.821
C07993=1193.263,54.011,-47.203,-179.284,5.819,148.820
C07994=1193.258,54.261,-47.219,-179.281,5.820,148.820
C07995=1193.253,54.529,-47.237,-179.278,5.821,148.819
C07996=1193.248,54.797,-47.254,-179.275,5.821,148.818
C07997=1193.242,55.067,-47.272,-179.273,5.823,148.818
C07998=1193.237,55.335,-47.289,-179.270,5.823,148.817
C07999=1193.231,55.584,-47.305,-179.267,5.824,148.817
C08000=1193.227,55.834,-47.322,-179.265,5.824,148.816
C08001=1193.222,56.082,-47.338,-179.262,5.826,148.816
C08002=1193.217,56.332,-47.354,-179.259,5.827,148.815
C08003=1193.212,56.582,-47.371,-179.257,5.827,148.814
C08004=1193.207,56.831,-47.387,-179.254,5.828,148.814
C08005=1193.202,57.081,-47.403,-179.251,5.830,148.813
C08006=1193.197,57.330,-47.420,-179.249,5.830,148.813
C08007=1193.192,57.579,-47.436,-179.246,5.831,148.812
C08008=1193.187,57.828,-47.453,-179.244,5.831,148.811
C08009=1193.182,58.078,-47.469,-179.242,5.832,148.811
C08010=1193.177,58.328,-47.486,-179.238,5.834,148.810
C08011=1193.172,58.577,-47.502,-179.236,5.834,148.810
C08012=1193.168,58.826,-47.519,-179.234,5.835,148.809
C08013=1193.162,59.076,-47.534,-179.231,5.836,148.809
C08014=1193.158,59.325,-47.551,-179.228,5.836,148.808
C08015=1193.153,59.575,-47.568,-179.226,5.838,148.807
C08016=1193.147,59.824,-47.585,-179.223,5.838,148.807
C08017=1193.143,60.074,-47.601,-179.220,5.839,148.806
C08018=1193.138,60.323,-47.617,-179.218,5.840,148.806
C08019=1193.132,60.572,-47.634,-179.216,5.840,148.805
C08020=1193.128,60.822,-47.651,-179.212,5.842,148.804
C08021=1193.123,61.071,-47.667,-179.210,5.843,148.804
C08022=1193.118,61.320,-47.684,-179.208,5.843,148.803
C08023=1193.112,61.570,-47.700,-179.206,5.844,148.803
C08024=1193.108,61.819,-47.717,-179.202,5.845,148.802
C08025=1193.103,62.069,-47.733,-179.200,5.846,148.802
C08026=1193.098,62.318,-47.750,-179.198,5.847,148.801
C08027=1193.093,62.567,-47.767,-179.195,5.847,148.800
C08028=1193.088,62.817,-47.784,-179.192,5.849,148.800
C08029=1193.083,63.066,-47.800,-179.190,5.850,148.799
C08030=1193.078,63.316,-47.817,-179.187,5.850,148.799
C08031=1193.074,63.565,-47.834,-179.185,5.851,148.798
C08032=1193.069,63.814,-47.850,-179.182,5.852,148.798
C08033=1193.063,64.064,-47.867,-179.179,5.853,148.797
C08034=1193.059,64.314,-47.883,-179.177,5.854,148.796
C08035=1193.054,64.562,-47.900,-179.174,5.854,148.796
C08036=1193.048,64.812,-47.917,-179.171,5.856,148.795
C08037=1193.044,65.062,-47.934,-179.169,5.857,148.795
C08038=1193.039,65.311,-47.950,-179.166,5.857,148.794
C08039=1193.034,65.560,-47.967,-179.164,5.858,148.794
C08040=1193.029,65.810,-47.984,-179.161,5.859,148.793
C08041=1193.025,66.059,-48.000,-179.158,5.860,148.792
C08042=1193.019,66.308,-48.017,-179.156,5.861,148.792
C08043=1193.014,66.558,-48.034,-179.153,5.861,148.791
C08044=1193.009,66.807,-48.052,-179.150,5.863,148.791
C08045=1193.004,67.056,-48.068,-179.148,5.864,148.790
C08046=1193.000,67.305,-48.085,-179.145,5.864,148.789
C08047=1192.995,67.555,-48.102,-179.143,5.865,148.789
C08048=1192.990,67.805,-48.119,-179.140,5.867,148.788
C08049=1192.984,68.054,-48.136,-179.137,5.867,148.788
C08050=1192.980,68.303,-48.153,-179.135,5.868,148.787
C08051=1192.975,68.553,-48.169,-179.133,5.869,148.787
C08052=1192.970,68.802,-48.186,-179.130,5.870,148.786
C08053=1192.965,69.051,-48.203,-179.127,5.871,148.786
C08054=1192.960,69.300,-48.221,-179.125,5.871,148.785
C08055=1192.956,69.550,-48.237,-179.123,5.872,148.784
C08056=1192.950,69.800,-48.255,-179.119,5.874,148.784
C08057=1192.946,70.049,-48.271,-179.117,5.874,148.783
C08058=1192.940,70.298,-48.288,-179.115,5.875,148.783
C08059=1192.936,70.548,-48.305,-179.111,5.876,148.782
C08060=1192.931,70.797,-48.323,-179.109,5.877,148.782
C08061=1192.926,71.046,-48.340,-179.107,5.878,148.781
C08062=1192.920,71.295,-48.356,-179.104,5.879,148.780
C08063=1192.916,71.545,-48.373,-179.101,5.880,148.780
C08064=1192.911,71.795,-48.390,-179.099,5.881,148.779
C08065=1192.907,72.044,-48.408,-179.096,5.882,148.779
C08066=1192.901,72.293,-48.425,-179.093,5.883,148.778
C08067=1192.897,72.543,-48.442,-179.091,5.884,148.778
C08068=1192.891,72.792,-48.459,-179.088,5.884,148.777
C08069=1192.886,73.041,-48.477,-179.086,5.885,148.776
C08070=1192.882,73.291,-48.493,-179.083,5.887,148.776
C08071=1192.876,73.540,-48.511,-179.080,5.887,148.775
C08072=1192.872,73.789,-48.528,-179.078,5.888,148.775
C08073=1192.866,74.038,-48.545,-179.075,5.889,148.774
C08074=1192.862,74.288,-48.561,-179.073,5.890,148.774
C08075=1192.857,74.538,-48.579,-179.070,5.891,148.773
C08076=1192.852,74.787,-48.597,-179.067,5.892,148.772
C08077=1192.847,75.036,-48.613,-179.065,5.893,148.772
C08078=1192.842,75.286,-48.631,-179.062,5.894,148.771
C08079=1192.838,75.535,-48.648,-179.060,5.895,148.771
C08080=1192.832,75.784,-48.665,-179.057,5.896,148.770
C08081=1192.827,76.033,-48.683,-179.054,5.897,148.770
C08082=1192.823,76.283,-48.700,-179.052,5.897,148.769
C08083=1192.818,76.533,-48.717,-179.049,5.899,148.769
C08084=1192.813,76.782,-48.735,-179.047,5.900,148.768
C08085=1192.808,77.031,-48.751,-179.044,5.900,148.767
C08086=1192.803,77.280,-48.769,-179.042,5.902,148.767
C08087=1192.798,77.530,-48.787,-179.039,5.903,148.766
C08088=1192.794,77.779,-48.804,-179.036,5.903,148.766
C08089=1192.789,78.029,-48.821,-179.034,5.905,148.765
C08090=1192.783,78.277,-48.839,-179.031,5.905,148.765
C08091=1192.779,78.527,-48.856,-179.029,5.906,148.764
C08092=1192.774,78.776,-48.874,-179.026,5.908,148.764
C08093=1192.768,79.026,-48.891,-179.023,5.909,148.763
C08094=1192.764,79.275,-48.909,-179.021,5.909,148.762
C08095=1192.759,79.524,-48.926,-179.018,5.911,148.762
C08096=1192.754,79.774,-48.944,-179.016,5.911,148.761
C08097=1192.749,80.023,-48.961,-179.013,5.912,148.761
C08098=1192.745,80.272,-48.978,-179.010,5.914,148.760
C08099=1192.739,80.541,-48.997,-179.008,5.914,148.760
C08100=1192.734,80.809,-49.016,-179.004,5.916,148.759
C08101=1192.728,81.078,-49.035,-179.002,5.916,148.759
C08102=1192.723,81.346,-49.053,-178.999,5.918,148.758
C08103=1192.718,81.596,-49.071,-178.996,5.918,148.757
C08104=1192.714,81.844,-49.089,-178.994,5.919,148.757
C08105=1192.709,82.094,-49.106,-178.991,5.921,148.756
C08106=1192.704,82.343,-49.124,-178.989,5.922,148.756
C08107=1192.699,82.593,-49.142,-178.986,5.923,148.755
C08108=1192.694,82.842,-49.159,-178.984,5.924,148.755
C08109=1192.689,83.091,-49.177,-178.981,5.924,148.754
C08110=1192.684,83.341,-49.194,-178.978,5.926,148.753
C08111=1192.679,83.590,-49.212,-178.976,5.927,148.753
C08112=1192.674,83.839,-49.230,-178.973,5.927,148.752
C08113=1192.669,84.089,-49.247,-178.970,5.929,148.752
C08114=1192.664,84.338,-49.265,-178.968,5.930,148.751
C08115=1192.660,84.587,-49.282,-178.965,5.930,148.751
C08116=1192.655,84.836,-49.300,-178.962,5.932,148.750
C08117=1192.650,85.086,-49.318,-178.960,5.933,148.750
C08118=1192.645,85.335,-49.336,-178.957,5.934,148.749
C08119=1192.640,85.585,-49.354,-178.955,5.935,148.749
C08120=1192.635,85.834,-49.372,-178.952,5.936,148.748
C08121=1192.630,86.084,-49.389,-178.949,5.937,148.748
C08122=1192.625,86.333,-49.407,-178.947,5.938,148.747
C08123=1192.620,86.582,-49.425,-178.944,5.938,148.746
C08124=1192.616,86.831,-49.442,-178.942,5.940,148.746
C08125=1192.611,87.081,-49.459,-178.939,5.941,148.745
C08126=1192.606,87.330,-49.477,-178.936,5.942,148.745
C08127=1192.601,87.579,-49.495,-178.934,5.943,148.744
C08128=1192.596,87.828,-49.513,-178.931,5.944,148.744
C08129=1192.592,88.078,-49.532,-178.928,5.945,148.743
C08130=1192.587,88.327,-49.550,-178.926,5.946,148.743
C08131=1192.582,88.577,-49.567,-178.923,5.947,148.742
C08132=1192.577,88.826,-49.585,-178.921,5.948,148.742
C08133=1192.572,89.075,-49.603,-178.918,5.949,148.741
C08134=1192.567,89.324,-49.621,-178.915,5.951,148.741
C08135=1192.562,89.574,-49.639,-178.913,5.951,148.740
C08136=1192.557,89.823,-49.657,-178.911,5.952,148.739
C08137=1192.552,90.072,-49.675,-178.907,5.954,148.739
C08138=1192.547,90.321,-49.693,-178.905,5.955,148.738
C08139=1192.543,90.571,-49.711,-178.902,5.956,148.738
C08140=1192.538,90.820,-49.729,-178.900,5.957,148.737
C08141=1192.533,91.069,-49.747,-178.897,5.957,148.737
C08142=1192.528,91.319,-49.764,-178.895,5.959,148.736
C08143=1192.523,91.568,-49.782,-178.892,5.960,148.736
C08144=1192.518,91.818,-49.800,-178.889,5.961,148.735
C08145=1192.513,92.067,-49.818,-178.887,5.962,148.735
C08146=1192.508,92.316,-49.836,-178.885,5.963,148.734
C08147=1192.504,92.566,-49.855,-178.881,5.964,148.733
C08148=1192.499,92.815,-49.873,-178.879,5.965,148.733
C08149=1192.494,93.064,-49.891,-178.876,5.967,148.732
C08150=1192.489,93.313,-49.910,-178.874,5.967,148.732
C08151=1192.484,93.562,-49.928,-178.871,5.969,148.731
C08152=1192.479,93.811,-49.946,-178.869,5.970,148.731
C08153=1192.475,94.061,-49.964,-178.866,5.970,148.730
C08154=1192.470,94.310,-49.982,-178.863,5.972,148.730
C08155=1192.465,94.560,-50.000,-178.861,5.973,148.729
C08156=1192.460,94.809,-50.018,-178.858,5.974,148.729
C08157=1192.455,95.058,-50.036,-178.855,5.975,148.728
C08158=1192.451,95.308,-50.055,-178.853,5.977,148.728
C08159=1192.445,95.557,-50.073,-178.850,5.977,148.727
C08160=1192.440,95.806,-50.091,-178.848,5.978,148.727
C08161=1192.435,96.055,-50.110,-178.845,5.980,148.726
C08162=1192.431,96.304,-50.128,-178.842,5.980,148.726
C08163=1192.426,96.554,-50.146,-178.839,5.982,148.725
C08164=1192.421,96.803,-50.164,-178.837,5.983,148.725
C08165=1192.416,97.053,-50.183,-178.834,5.984,148.724
C08166=1192.411,97.302,-50.201,-178.832,5.985,148.724
C08167=1192.407,97.551,-50.220,-178.829,5.986,148.723
C08168=1192.402,97.800,-50.238,-178.827,5.987,148.722
C08169=1192.397,98.050,-50.256,-178.824,5.988,148.722
C08170=1192.391,98.299,-50.274,-178.821,5.990,148.721
C08171=1192.387,98.549,-50.293,-178.819,5.990,148.721
C08172=1192.382,98.797,-50.311,-178.816,5.992,148.720
C08173=1192.377,99.047,-50.329,-178.814,5.993,148.720
C08174=1192.372,99.296,-50.348,-178.811,5.994,148.719
C08175=1192.368,99.545,-50.367,-178.808,5.995,148.719
C08176=1192.363,99.795,-50.385,-178.805,5.997,148.718
C08177=1192.358,100.044,-50.403,-178.803,5.997,148.718
C08178=1192.352,100.293,-50.421,-178.800,5.998,148.717
C08179=1192.348,100.542,-50.440,-178.798,6.000,148.717
C08180=1192.343,100.792,-50.458,-178.795,6.000,148.716
C08181=1192.339,101.041,-50.476,-178.792,6.002,148.716
C08182=1192.334,101.290,-50.496,-178.790,6.003,148.715
C08183=1192.329,101.540,-50.514,-178.787,6.004,148.715
C08184=1192.324,101.789,-50.532,-178.784,6.005,148.714
C08185=1192.319,102.038,-50.552,-178.782,6.007,148.714
C08186=1192.314,102.287,-50.570,-178.780,6.008,148.713
C08187=1192.310,102.536,-50.588,-178.776,6.009,148.713
C08188=1192.305,102.786,-50.607,-178.774,6.010,148.712
C08189=1192.300,103.035,-50.625,-178.771,6.011,148.711
C08190=1192.295,103.284,-50.644,-178.769,6.012,148.711
C08191=1192.290,103.534,-50.663,-178.766,6.014,148.710
C08192=1192.285,103.783,-50.682,-178.764,6.015,148.710
C08193=1192.281,104.032,-50.700,-178.760,6.016,148.709
C08194=1192.276,104.281,-50.719,-178.758,6.017,148.709
C08195=1192.271,104.531,-50.737,-178.756,6.019,148.709
C08196=1192.266,104.779,-50.757,-178.753,6.019,148.708
C08197=1192.261,105.029,-50.775,-178.751,6.020,148.707
C08198=1192.257,105.278,-50.794,-178.748,6.022,148.707
C08199=1192.251,105.527,-50.812,-178.746,6.022,148.706
C08200=1192.247,105.777,-50.831,-178.742,6.024,148.706
C08201=1192.241,106.026,-50.850,-178.740,6.025,148.705
C08202=1192.237,106.275,-50.869,-178.737,6.026,148.705
C08203=1192.232,106.544,-50.889,-178.734,6.028,148.704
C08204=1192.227,106.812,-50.909,-178.732,6.028,148.704
C08205=1192.222,107.081,-50.929,-178.729,6.030,148.703
C08206=1192.216,107.349,-50.949,-178.726,6.032,148.703
C08207=1192.211,107.598,-50.968,-178.724,6.033,148.702
C08208=1192.206,107.848,-50.988,-178.721,6.034,148.702
C08209=1192.201,108.097,-51.006,-178.718,6.035,148.701
C08210=1192.197,108.346,-51.025,-178.715,6.036,148.701
C08211=1192.192,108.595,-51.043,-178.713,6.037,148.700
C08212=1192.188,108.845,-51.062,-178.710,6.039,148.700
C08213=1192.182,109.094,-51.082,-178.708,6.039,148.699
C08214=1192.178,109.343,-51.100,-178.705,6.041,148.699
C08215=1192.173,109.592,-51.119,-178.702,6.042,148.698
C08216=1192.167,109.841,-51.139,-178.700,6.044,148.698
C08217=1192.163,110.091,-51.157,-178.697,6.044,148.697
C08218=1192.158,110.340,-51.176,-178.694,6.046,148.697
C08219=1192.154,110.589,-51.195,-178.692,6.047,148.696
C08220=1192.148,110.838,-51.215,-178.689,6.048,148.696
C08221=1192.144,111.088,-51.233,-178.686,6.050,148.695
C08222=1192.139,111.337,-51.252,-178.684,6.051,148.695
C08223=1192.135,111.586,-51.271,-178.681,6.052,148.694
C08224=1192.129,111.835,-51.291,-178.679,6.053,148.694
C08225=1192.124,112.085,-51.310,-178.676,6.055,148.693
C08226=1192.120,112.334,-51.328,-178.674,6.056,148.693
C08227=1192.115,112.583,-51.348,-178.670,6.057,148.692
C08228=1192.110,112.832,-51.367,-178.668,6.058,148.692
C08229=1192.105,113.082,-51.385,-178.666,6.060,148.691
C08230=1192.100,113.331,-51.405,-178.663,6.060,148.691
C08231=1192.096,113.580,-51.424,-178.660,6.062,148.690
C08232=1192.091,113.829,-51.443,-178.658,6.062,148.690
C08233=1192.086,114.079,-51.463,-178.655,6.064,148.689
C08234=1192.081,114.327,-51.481,-178.652,6.066,148.689
C08235=1192.077,114.577,-51.501,-178.650,6.067,148.688
C08236=1192.071,114.826,-51.520,-178.647,6.068,148.688
C08237=1192.067,115.075,-51.539,-178.644,6.069,148.687
C08238=1192.062,115.324,-51.558,-178.642,6.071,148.687
C08239=1192.057,115.574,-51.578,-178.640,6.072,148.686
C08240=1192.052,115.822,-51.596,-178.636,6.073,148.686
C08241=1192.047,116.072,-51.616,-178.634,6.074,148.685
C08242=1192.042,116.321,-51.635,-178.632,6.076,148.685
C08243=1192.038,116.570,-51.654,-178.628,6.077,148.684
C08244=1192.033,116.820,-51.674,-178.626,6.078,148.684
C08245=1192.028,117.069,-51.693,-178.623,6.079,148.683
C08246=1192.023,117.318,-51.713,-178.621,6.080,148.683
C08247=1192.019,117.567,-51.732,-178.618,6.082,148.682
C08248=1192.014,117.816,-51.751,-178.616,6.083,148.682
C08249=1192.009,118.066,-51.771,-178.613,6.084,148.681
C08250=1192.004,118.315,-51.790,-178.610,6.086,148.681
C08251=1192.000,118.564,-51.809,-178.608,6.087,148.680
C08252=1191.995,118.813,-51.829,-178.605,6.089,148.680
C08253=1191.990,119.062,-51.848,-178.602,6.089,148.679
C08254=1191.985,119.312,-51.868,-178.600,6.091,148.679
C08255=1191.980,119.561,-51.887,-178.597,6.092,148.678
C08256=1191.976,119.810,-51.906,-178.594,6.093,148.678
C08257=1191.970,120.059,-51.926,-178.592,6.095,148.677
C08258=1191.966,120.309,-51.945,-178.589,6.096,148.677
C08259=1191.961,120.558,-51.965,-178.586,6.097,148.676
C08260=1191.956,120.807,-51.984,-178.584,6.098,148.676
C08261=1191.952,121.056,-52.003,-178.581,6.100,148.676
C08262=1191.947,121.305,-52.024,-178.578,6.101,148.675
C08263=1191.942,121.554,-52.043,-178.576,6.102,148.675
C08264=1191.937,121.804,-52.063,-178.573,6.104,148.674
C08265=1191.932,122.053,-52.082,-178.571,6.105,148.674
C08266=1191.927,122.302,-52.102,-178.568,6.106,148.673
C08267=1191.923,122.551,-52.121,-178.565,6.108,148.673
C08268=1191.918,122.800,-52.141,-178.563,6.109,148.672
C08269=1191.913,123.049,-52.160,-178.560,6.110,148.672
C08270=1191.908,123.299,-52.180,-178.558,6.111,148.671
C08271=1191.904,123.548,-52.200,-178.555,6.113,148.671
C08272=1191.899,123.796,-52.220,-178.552,6.115,148.670
C08273=1191.894,124.046,-52.239,-178.550,6.116,148.670
C08274=1191.889,124.296,-52.259,-178.547,6.117,148.669
C08275=1191.884,124.544,-52.278,-178.545,6.118,148.669
C08276=1191.879,124.793,-52.299,-178.542,6.120,148.668
C08277=1191.875,125.043,-52.318,-178.539,6.121,148.668
C08278=1191.870,125.293,-52.338,-178.537,6.122,148.667
C08279=1191.865,125.541,-52.357,-178.534,6.124,148.667
C08280=1191.861,125.790,-52.377,-178.531,6.125,148.666
C08281=1191.856,126.040,-52.397,-178.529,6.126,148.666
C08282=1191.851,126.289,-52.416,-178.526,6.128,148.666
C08283=1191.846,126.537,-52.436,-178.523,6.128,148.665
C08284=1191.842,126.787,-52.456,-178.521,6.130,148.665
C08285=1191.837,127.037,-52.476,-178.518,6.132,148.664
C08286=1191.832,127.286,-52.496,-178.515,6.133,148.664
C08287=1191.827,127.534,-52.515,-178.513,6.134,148.663
C08288=1191.823,127.783,-52.536,-178.510,6.136,148.663
C08289=1191.818,128.033,-52.555,-178.507,6.137,148.662
C08290=1191.813,128.283,-52.575,-178.505,6.138,148.662
C08291=1191.808,128.531,-52.595,-178.503,6.139,148.661
C08292=1191.803,128.780,-52.615,-178.499,6.141,148.661
C08293=1191.799,129.029,-52.635,-178.497,6.142,148.660
C08294=1191.793,129.279,-52.655,-178.495,6.143,148.660
C08295=1191.789,129.528,-52.676,-178.492,6.145,148.660
C08296=1191.784,129.777,-52.695,-178.489,6.147,148.659
C08297=1191.779,130.026,-52.715,-178.487,6.148,148.659
C08298=1191.774,130.275,-52.735,-178.484,6.149,148.658
C08299=1191.770,130.524,-52.755,-178.481,6.151,148.658
C08300=1191.765,130.774,-52.775,-178.479,6.152,148.657
C08301=1191.760,131.022,-52.795,-178.476,6.153,148.657
C08302=1191.755,131.272,-52.815,-178.473,6.155,148.656
C08303=1191.751,131.521,-52.835,-178.471,6.156,148.656
C08304=1191.746,131.771,-52.855,-178.468,6.158,148.655
C08305=1191.741,132.020,-52.876,-178.465,6.159,148.655
C08306=1191.736,132.269,-52.895,-178.463,6.160,148.654
C08307=1191.732,132.537,-52.917,-178.460,6.162,148.654
C08308=1191.726,132.806,-52.939,-178.457,6.163,148.653
C08309=1191.721,133.074,-52.961,-178.454,6.165,148.653
C08310=1191.716,133.343,-52.982,-178.451,6.166,148.652
C08311=1191.711,133.592,-53.003,-178.449,6.167,148.652
C08312=1191.707,133.842,-53.022,-178.446,6.169,148.651
C08313=1191.701,134.090,-53.043,-178.443,6.171,148.651
C08314=1191.696,134.339,-53.063,-178.441,6.171,148.650
C08315=1191.692,134.589,-53.083,-178.438,6.173,148.650
C08316=1191.687,134.838,-53.103,-178.435,6.175,148.650
C08317=1191.683,135.087,-53.124,-178.433,6.177,148.649
C08318=1191.677,135.337,-53.144,-178.430,6.177,148.649
C08319=1191.673,135.585,-53.164,-178.427,6.179,148.648
C08320=1191.668,135.834,-53.185,-178.425,6.181,148.648
C08321=1191.664,136.083,-53.205,-178.422,6.181,148.647
C08322=1191.659,136.333,-53.225,-178.420,6.183,148.647
C08323=1191.654,136.581,-53.245,-178.417,6.185,148.647
C08324=1191.649,136.830,-53.266,-178.415,6.186,148.646
C08325=1191.645,137.079,-53.286,-178.412,6.187,148.645
C08326=1191.639,137.329,-53.306,-178.409,6.189,148.645
C08327=1191.635,137.578,-53.327,-178.407,6.190,148.645
C08328=1191.630,137.827,-53.347,-178.404,6.192,148.644
C08329=1191.625,138.076,-53.368,-178.401,6.193,148.644
C08330=1191.621,138.325,-53.388,-178.398,6.195,148.643
C08331=1191.616,138.575,-53.408,-178.396,6.196,148.643
C08332=1191.611,138.824,-53.429,-178.393,6.198,148.643
C08333=1191.606,139.073,-53.449,-178.390,6.199,148.642
C08334=1191.602,139.322,-53.470,-178.388,6.200,148.642
C08335=1191.597,139.571,-53.491,-178.385,6.202,148.641
C08336=1191.592,139.820,-53.511,-178.383,6.203,148.641
C08337=1191.588,140.069,-53.531,-178.380,6.205,148.640
C08338=1191.583,140.319,-53.552,-178.377,6.206,148.640
C08339=1191.578,140.567,-53.573,-178.375,6.208,148.639
C08340=1191.574,140.816,-53.593,-178.372,6.209,148.639
C08341=1191.568,141.066,-53.613,-178.370,6.210,148.639
C08342=1191.564,141.315,-53.634,-178.367,6.212,148.638
C08343=1191.559,141.565,-53.655,-178.364,6.214,148.638
C08344=1191.554,141.813,-53.675,-178.361,6.215,148.637
C08345=1191.550,142.062,-53.695,-178.359,6.216,148.637
C08346=1191.545,142.312,-53.716,-178.356,6.218,148.636
C08347=1191.540,142.561,-53.737,-178.353,6.219,148.636
C08348=1191.535,142.810,-53.758,-178.351,6.221,148.635
C08349=1191.531,143.059,-53.778,-178.349,6.222,148.635
C08350=1191.525,143.308,-53.799,-178.345,6.224,148.634
C08351=1191.521,143.557,-53.819,-178.343,6.225,148.634
C08352=1191.516,143.806,-53.840,-178.341,6.226,148.634
C08353=1191.512,144.055,-53.862,-178.338,6.228,148.633
C08354=1191.507,144.304,-53.882,-178.335,6.230,148.633
C08355=1191.502,144.553,-53.903,-178.332,6.231,148.632
C08356=1191.498,144.802,-53.923,-178.330,6.232,148.632
C08357=1191.493,145.052,-53.945,-178.327,6.234,148.631
C08358=1191.489,145.301,-53.965,-178.325,6.236,148.631
C08359=1191.483,145.550,-53.986,-178.322,6.237,148.631
C08360=1191.479,145.799,-54.006,-178.319,6.238,148.630
C08361=1191.474,146.048,-54.027,-178.317,6.240,148.630
C08362=1191.469,146.297,-54.049,-178.314,6.242,148.629
C08363=1191.465,146.546,-54.069,-178.311,6.243,148.629
C08364=1191.459,146.795,-54.090,-178.309,6.245,148.629
C08365=1191.455,147.044,-54.111,-178.306,6.246,148.628
C08366=1191.450,147.293,-54.132,-178.303,6.248,148.628
C08367=1191.446,147.542,-54.153,-178.301,6.249,148.627
C08368=1191.441,147.791,-54.174,-178.298,6.251,148.627
C08369=1191.436,148.041,-54.195,-178.296,6.252,148.626
C08370=1191.431,148.290,-54.215,-178.293,6.253,148.626
C08371=1191.427,148.538,-54.237,-178.290,6.255,148.625
C08372=1191.422,148.787,-54.257,-178.287,6.257,148.625
C08373=1191.417,149.037,-54.278,-178.285,6.258,148.625
C08374=1191.412,149.286,-54.299,-178.282,6.260,148.624
C08375=1191.408,149.535,-54.321,-178.280,6.262,148.624
C08376=1191.403,149.784,-54.342,-178.277,6.263,148.623
C08377=1191.399,150.033,-54.362,-178.274,6.265,148.623
C08378=1191.394,150.282,-54.384,-178.272,6.266,148.623
C08379=1191.389,150.531,-54.405,-178.269,6.267,148.622
C08380=1191.384,150.780,-54.425,-178.266,6.269,148.622
C08381=1191.380,151.029,-54.447,-178.263,6.271,148.621
C08382=1191.375,151.279,-54.468,-178.261,6.272,148.621
C08383=1191.370,151.528,-54.489,-178.258,6.273,148.620
C08384=1191.365,151.776,-54.510,-178.256,6.275,148.620
C08385=1191.360,152.025,-54.531,-178.253,6.277,148.620
C08386=1191.356,152.275,-54.553,-178.250,6.279,148.619
C08387=1191.352,152.524,-54.574,-178.248,6.280,148.619
C08388=1191.346,152.773,-54.595,-178.245,6.281,148.618
C08389=1191.341,153.022,-54.616,-178.242,6.283,148.618
C08390=1191.336,153.271,-54.637,-178.240,6.285,148.618
C08391=1191.333,153.520,-54.659,-178.237,6.286,148.617
C08392=1191.328,153.769,-54.680,-178.235,6.287,148.617
C08393=1191.323,154.018,-54.701,-178.232,6.289,148.616
C08394=1191.318,154.267,-54.722,-178.229,6.291,148.616
C08395=1191.314,154.516,-54.744,-178.226,6.292,148.615
C08396=1191.309,154.765,-54.765,-178.224,6.294,148.615
C08397=1191.304,155.014,-54.786,-178.221,6.296,148.615
C08398=1191.299,155.263,-54.807,-178.219,6.297,148.614
C08399=1191.295,155.513,-54.829,-178.216,6.299,148.614
C08400=1191.290,155.761,-54.850,-178.214,6.300,148.614
C08401=1191.285,156.010,-54.871,-178.210,6.302,148.613
C08402=1191.280,156.259,-54.893,-178.208,6.304,148.613
C08403=1191.276,156.509,-54.914,-178.206,6.305,148.612
C08404=1191.271,156.757,-54.936,-178.203,6.306,148.612
C08405=1191.266,157.007,-54.957,-178.200,6.308,148.611
C08406=1191.262,157.256,-54.979,-178.198,6.310,148.611
C08407=1191.257,157.504,-55.000,-178.195,6.312,148.611
C08408=1191.252,157.754,-55.021,-178.192,6.313,148.610
C08409=1191.248,158.003,-55.043,-178.190,6.314,148.610
C08410=1191.243,158.252,-55.065,-178.187,6.316,148.609
C08411=1191.238,158.521,-55.088,-178.184,6.318,148.609
C08412=1191.233,158.790,-55.111,-178.182,6.319,148.609
C08413=1191.228,159.059,-55.134,-178.178,6.322,148.608
C08414=1191.223,159.328,-55.158,-178.175,6.323,148.608
C08415=1191.218,159.577,-55.179,-178.173,6.324,148.607
C08416=1191.213,159.826,-55.201,-178.170,6.326,148.607
C08417=1191.209,160.075,-55.223,-178.168,6.328,148.606
C08418=1191.204,160.324,-55.244,-178.165,6.330,148.606
C08419=1191.199,160.573,-55.265,-178.162,6.332,148.606
C08420=1191.194,160.822,-55.287,-178.159,6.333,148.605
C08421=1191.189,161.071,-55.309,-178.157,6.335,148.605
C08422=1191.185,161.319,-55.330,-178.154,6.336,148.604
C08423=1191.181,161.569,-55.352,-178.152,6.337,148.604
C08424=1191.176,161.818,-55.373,-178.149,6.339,148.604
C08425=1191.172,162.067,-55.395,-178.146,6.341,148.603
C08426=1191.167,162.316,-55.417,-178.144,6.343,148.603
C08427=1191.162,162.564,-55.439,-178.141,6.345,148.603
C08428=1191.158,162.814,-55.461,-178.138,6.346,148.602
C08429=1191.153,163.062,-55.482,-178.136,6.347,148.602
C08430=1191.148,163.312,-55.504,-178.133,6.349,148.601
C08431=1191.142,163.561,-55.526,-178.130,6.351,148.601
C08432=1191.138,163.810,-55.548,-178.128,6.352,148.600
C08433=1191.133,164.059,-55.570,-178.125,6.354,148.600
C08434=1191.128,164.308,-55.591,-178.122,6.356,148.600
C08435=1191.124,164.557,-55.613,-178.120,6.358,148.599
C08436=1191.119,164.806,-55.635,-178.117,6.359,148.599
C08437=1191.115,165.055,-55.657,-178.115,6.360,148.599
C08438=1191.110,165.304,-55.679,-178.112,6.362,148.598
C08439=1191.105,165.553,-55.700,-178.110,6.364,148.598
C08440=1191.101,165.802,-55.722,-178.107,6.366,148.597
C08441=1191.096,166.050,-55.744,-178.104,6.368,148.597
C08442=1191.092,166.300,-55.766,-178.102,6.369,148.597
C08443=1191.087,166.548,-55.788,-178.098,6.371,148.596
C08444=1191.082,166.798,-55.811,-178.096,6.373,148.596
C08445=1191.077,167.047,-55.832,-178.093,6.374,148.595
C08446=1191.073,167.296,-55.854,-178.090,6.376,148.595
C08447=1191.068,167.545,-55.876,-178.088,6.377,148.595
C08448=1191.064,167.794,-55.898,-178.086,6.379,148.594
C08449=1191.059,168.043,-55.920,-178.083,6.381,148.594
C08450=1191.054,168.292,-55.942,-178.080,6.382,148.594
C08451=1191.049,168.540,-55.965,-178.078,6.384,148.593
C08452=1191.045,168.790,-55.987,-178.075,6.386,148.593
C08453=1191.040,169.038,-56.008,-178.072,6.388,148.592
C08454=1191.036,169.288,-56.030,-178.070,6.390,148.592
C08455=1191.030,169.537,-56.053,-178.067,6.391,148.592
C08456=1191.026,169.786,-56.075,-178.064,6.393,148.591
C08457=1191.021,170.035,-56.097,-178.062,6.395,148.591
C08458=1191.017,170.283,-56.119,-178.059,6.396,148.591
C08459=1191.012,170.532,-56.141,-178.057,6.398,148.590
C08460=1191.007,170.782,-56.164,-178.054,6.400,148.590
C08461=1191.002,171.030,-56.185,-178.051,6.401,148.589
C08462=1190.998,171.280,-56.207,-178.048,6.403,148.589
C08463=1190.994,171.529,-56.231,-178.046,6.405,148.589
C08464=1190.989,171.777,-56.252,-178.043,6.406,148.588
C08465=1190.984,172.027,-56.274,-178.040,6.408,148.588
C08466=1190.980,172.275,-56.296,-178.038,6.410,148.587
C08467=1190.975,172.524,-56.319,-178.035,6.412,148.587
C08468=1190.970,172.773,-56.341,-178.032,6.413,148.587
C08469=1190.966,173.022,-56.363,-178.030,6.415,148.586
C08470=1190.961,173.271,-56.387,-178.027,6.417,148.586
C08471=1190.956,173.520,-56.408,-178.024,6.419,148.586
C08472=1190.952,173.769,-56.430,-178.022,6.420,148.585
C08473=1190.947,174.018,-56.453,-178.019,6.422,148.585
C08474=1190.942,174.267,-56.475,-178.017,6.423,148.585
C08475=1190.938,174.516,-56.497,-178.014,6.425,148.584
C08476=1190.933,174.765,-56.520,-178.011,6.427,148.584
C08477=1190.928,175.014,-56.542,-178.009,6.429,148.583
C08478=1190.924,175.263,-56.564,-178.006,6.431,148.583
C08479=1190.919,175.512,-56.587,-178.003,6.432,148.583
C08480=1190.915,175.761,-56.609,-178.001,6.434,148.582
C08481=1190.909,176.009,-56.632,-177.998,6.436,148.582
C08482=1190.905,176.259,-56.655,-177.995,6.438,148.582
C08483=1190.901,176.507,-56.677,-177.993,6.439,148.581
C08484=1190.895,176.756,-56.700,-177.990,6.441,148.581
C08485=1190.891,177.005,-56.722,-177.987,6.443,148.581
C08486=1190.886,177.255,-56.745,-177.985,6.445,148.580
C08487=1190.882,177.503,-56.767,-177.982,6.447,148.580
C08488=1190.877,177.752,-56.790,-177.979,6.448,148.579
C08489=1190.873,178.001,-56.813,-177.977,6.450,148.579
C08490=1190.867,178.250,-56.835,-177.974,6.452,148.579
C08491=1190.863,178.499,-56.858,-177.971,6.454,148.578
C08492=1190.858,178.748,-56.880,-177.969,6.456,148.578
C08493=1190.854,178.996,-56.903,-177.966,6.457,148.578
C08494=1190.849,179.246,-56.926,-177.963,6.459,148.577
C08495=1190.845,179.495,-56.948,-177.961,6.461,148.577
C08496=1190.840,179.744,-56.972,-177.958,6.463,148.577
C08497=1190.835,179.993,-56.993,-177.955,6.465,148.576
C08498=1190.831,180.242,-57.017,-177.953,6.466,148.576
C08499=1190.826,180.491,-57.039,-177.950,6.468,148.576
C08500=1190.822,180.740,-57.062,-177.947,6.470,148.575
C08501=1190.817,180.988,-57.084,-177.945,6.472,148.575
C08502=1190.812,181.238,-57.107,-177.942,6.474,148.574
C08503=1190.808,181.486,-57.130,-177.939,6.475,148.574
C08504=1190.803,181.735,-57.153,-177.937,6.477,148.574
C08505=1190.799,181.984,-57.175,-177.935,6.479,148.574
C08506=1190.794,182.233,-57.198,-177.932,6.481,148.573
C08507=1190.789,182.482,-57.222,-177.929,6.483,148.573
C08508=1190.785,182.731,-57.244,-177.927,6.485,148.573
C08509=1190.780,182.980,-57.267,-177.924,6.486,148.572
C08510=1190.776,183.228,-57.289,-177.921,6.488,148.572
C08511=1190.771,183.477,-57.313,-177.919,6.490,148.571
C08512=1190.766,183.727,-57.336,-177.916,6.492,148.571
C08513=1190.761,183.975,-57.358,-177.913,6.494,148.571
C08514=1190.757,184.224,-57.381,-177.911,6.495,148.570
C08515=1190.751,184.494,-57.406,-177.908,6.497,148.570
C08516=1190.747,184.763,-57.431,-177.905,6.499,148.570
C08517=1190.742,185.033,-57.456,-177.903,6.501,148.569
C08518=1190.737,185.302,-57.481,-177.899,6.503,148.569
C08519=1190.732,185.551,-57.504,-177.897,6.505,148.569
C08520=1190.727,185.801,-57.527,-177.894,6.507,148.568
C08521=1190.723,186.049,-57.550,-177.891,6.509,148.568
C08522=1190.719,186.298,-57.573,-177.889,6.511,148.568
C08523=1190.713,186.547,-57.596,-177.886,6.512,148.567
C08524=1190.709,186.796,-57.619,-177.883,6.514,148.567
C08525=1190.705,187.045,-57.642,-177.881,6.516,148.567
C08526=1190.700,187.294,-57.665,-177.878,6.518,148.566
C08527=1190.695,187.543,-57.689,-177.875,6.520,148.566
C08528=1190.691,187.792,-57.712,-177.873,6.521,148.565
C08529=1190.687,188.040,-57.735,-177.870,6.523,148.565
C08530=1190.681,188.289,-57.758,-177.867,6.525,148.565
C08531=1190.677,188.538,-57.781,-177.865,6.527,148.565
C08532=1190.672,188.787,-57.805,-177.862,6.529,148.564
C08533=1190.668,189.035,-57.827,-177.860,6.531,148.564
C08534=1190.663,189.285,-57.851,-177.857,6.533,148.564
C08535=1190.659,189.534,-57.874,-177.854,6.534,148.563
C08536=1190.654,189.783,-57.898,-177.852,6.536,148.563
C08537=1190.649,190.032,-57.921,-177.849,6.538,148.562
C08538=1190.645,190.281,-57.944,-177.846,6.540,148.562
C08539=1190.640,190.529,-57.967,-177.843,6.542,148.562
C08540=1190.635,190.778,-57.990,-177.841,6.544,148.561
C08541=1190.631,191.027,-58.013,-177.838,6.546,148.561
C08542=1190.626,191.276,-58.037,-177.836,6.548,148.561
C08543=1190.621,191.525,-58.060,-177.833,6.550,148.561
C08544=1190.617,191.773,-58.084,-177.830,6.552,148.560
C08545=1190.612,192.022,-58.107,-177.828,6.553,148.560
C08546=1190.607,192.271,-58.131,-177.825,6.555,148.560
C08547=1190.603,192.520,-58.154,-177.822,6.557,148.559
C08548=1190.599,192.769,-58.177,-177.820,6.559,148.559
C08549=1190.594,193.018,-58.200,-177.817,6.561,148.559
C08550=1190.590,193.266,-58.224,-177.814,6.562,148.558
C08551=1190.585,193.515,-58.248,-177.812,6.565,148.558
C08552=1190.580,193.765,-58.271,-177.810,6.566,148.558
C08553=1190.576,194.014,-58.294,-177.806,6.569,148.557
C08554=1190.571,194.263,-58.318,-177.804,6.571,148.557
C08555=1190.566,194.511,-58.342,-177.801,6.573,148.557
C08556=1190.562,194.760,-58.365,-177.798,6.574,148.556
C08557=1190.557,195.009,-58.389,-177.796,6.576,148.556
C08558=1190.553,195.257,-58.413,-177.793,6.578,148.556
C08559=1190.548,195.507,-58.436,-177.791,6.580,148.555
C08560=1190.543,195.756,-58.459,-177.788,6.582,148.555
C08561=1190.539,196.004,-58.484,-177.786,6.584,148.555
C08562=1190.534,196.253,-58.507,-177.783,6.586,148.554
C08563=1190.529,196.502,-58.530,-177.780,6.587,148.554
C08564=1190.525,196.750,-58.554,-177.777,6.590,148.554
C08565=1190.520,196.999,-58.578,-177.774,6.592,148.553
C08566=1190.516,197.249,-58.601,-177.772,6.594,148.553
C08567=1190.511,197.497,-58.625,-177.769,6.596,148.553
C08568=1190.507,197.746,-58.648,-177.767,6.598,148.553
C08569=1190.502,197.994,-58.673,-177.764,6.599,148.552
C08570=1190.497,198.243,-58.696,-177.762,6.601,148.552
C08571=1190.493,198.492,-58.719,-177.759,6.603,148.552
C08572=1190.488,198.741,-58.743,-177.756,6.605,148.551
C08573=1190.484,198.990,-58.767,-177.753,6.608,148.551
C08574=1190.479,199.238,-58.791,-177.751,6.610,148.551
C08575=1190.474,199.488,-58.815,-177.748,6.611,148.550
C08576=1190.470,199.737,-58.839,-177.745,6.613,148.550
C08577=1190.465,199.986,-58.863,-177.743,6.615,148.550
C08578=1190.461,200.234,-58.887,-177.740,6.617,148.549
C08579=1190.456,200.483,-58.910,-177.738,6.619,148.549
C08580=1190.452,200.732,-58.934,-177.735,6.621,148.549
C08581=1190.447,200.981,-58.957,-177.733,6.623,148.549
C08582=1190.443,201.229,-58.981,-177.729,6.625,148.548
C08583=1190.438,201.478,-59.006,-177.727,6.627,148.548
C08584=1190.433,201.727,-59.029,-177.724,6.629,148.548
C08585=1190.429,201.976,-59.054,-177.722,6.631,148.547
C08586=1190.424,202.225,-59.077,-177.719,6.633,148.547
C08587=1190.420,202.473,-59.101,-177.717,6.634,148.547
C08588=1190.415,202.722,-59.126,-177.714,6.636,148.546
C08589=1190.410,202.971,-59.149,-177.711,6.639,148.546
C08590=1190.406,203.220,-59.173,-177.709,6.641,148.546
C08591=1190.401,203.468,-59.198,-177.706,6.643,148.546
C08592=1190.397,203.718,-59.221,-177.703,6.645,148.545
C08593=1190.392,203.966,-59.246,-177.701,6.646,148.545
C08594=1190.388,204.215,-59.270,-177.698,6.648,148.545
C08595=1190.383,204.464,-59.293,-177.696,6.650,148.544
C08596=1190.379,204.712,-59.317,-177.693,6.653,148.544
C08597=1190.374,204.962,-59.342,-177.690,6.655,148.544
C08598=1190.370,205.210,-59.367,-177.687,6.657,148.544
C08599=1190.365,205.459,-59.390,-177.685,6.659,148.543
C08600=1190.360,205.708,-59.415,-177.682,6.661,148.543
C08601=1190.356,205.956,-59.439,-177.680,6.662,148.543
C08602=1190.352,206.205,-59.463,-177.676,6.665,148.542
C08603=1190.347,206.454,-59.488,-177.674,6.667,148.542
C08604=1190.342,206.703,-59.511,-177.671,6.669,148.542
C08605=1190.338,206.952,-59.535,-177.669,6.671,148.542
C08606=1190.332,207.200,-59.560,-177.666,6.673,148.541
C08607=1190.329,207.449,-59.584,-177.664,6.674,148.541
C08608=1190.324,207.698,-59.608,-177.660,6.677,148.541
C08609=1190.319,207.947,-59.633,-177.658,6.679,148.540
C08610=1190.314,208.196,-59.656,-177.656,6.681,148.540
C08611=1190.311,208.445,-59.681,-177.653,6.683,148.540
C08612=1190.305,208.693,-59.706,-177.650,6.685,148.539
C08613=1190.301,208.942,-59.730,-177.647,6.687,148.539
C08614=1190.296,209.191,-59.754,-177.645,6.689,148.539
C08615=1190.292,209.440,-59.779,-177.642,6.691,148.539
C08616=1190.288,209.688,-59.803,-177.640,6.693,148.538
C08617=1190.283,209.937,-59.827,-177.637,6.695,148.538
C08618=1190.279,210.186,-59.852,-177.635,6.697,148.538
C08619=1190.274,210.456,-59.879,-177.632,6.700,148.538
C08620=1190.269,210.726,-59.905,-177.629,6.701,148.537
C08621=1190.263,210.997,-59.931,-177.626,6.704,148.537
C08622=1190.259,211.268,-59.958,-177.623,6.706,148.537
C08623=1190.254,211.516,-59.982,-177.620,6.709,148.536
C08624=1190.249,211.765,-60.007,-177.617,6.710,148.536
C08625=1190.245,212.014,-60.032,-177.615,6.713,148.536
C08626=1190.240,212.263,-60.056,-177.612,6.714,148.535
C08627=1190.236,212.511,-60.081,-177.610,6.716,148.535
C08628=1190.231,212.760,-60.106,-177.606,6.719,148.535
C08629=1190.227,213.009,-60.130,-177.604,6.721,148.535
C08630=1190.222,213.257,-60.155,-177.602,6.723,148.534
C08631=1190.218,213.506,-60.179,-177.599,6.725,148.534
C08632=1190.213,213.755,-60.204,-177.597,6.727,148.534
C08633=1190.209,214.003,-60.228,-177.594,6.729,148.534
C08634=1190.204,214.253,-60.253,-177.591,6.731,148.533
C08635=1190.199,214.501,-60.278,-177.588,6.733,148.533
C08636=1190.195,214.749,-60.302,-177.586,6.735,148.533
C08637=1190.190,214.999,-60.328,-177.583,6.738,148.533
C08638=1190.186,215.247,-60.352,-177.580,6.740,148.532
C08639=1190.181,215.497,-60.377,-177.578,6.741,148.532
C08640=1190.177,215.745,-60.402,-177.575,6.744,148.532
C08641=1190.172,215.993,-60.426,-177.573,6.745,148.531
C08642=1190.168,216.243,-60.451,-177.570,6.748,148.531
C08643=1190.163,216.491,-60.475,-177.567,6.750,148.531
C08644=1190.159,216.740,-60.501,-177.565,6.752,148.531
C08645=1190.154,216.989,-60.526,-177.562,6.754,148.530
C08646=1190.150,217.237,-60.550,-177.559,6.756,148.530
C08647=1190.145,217.486,-60.575,-177.557,6.759,148.530
C08648=1190.140,217.735,-60.600,-177.554,6.760,148.530
C08649=1190.136,217.984,-60.625,-177.551,6.762,148.529
C08650=1190.132,218.232,-60.650,-177.549,6.765,148.529
C08651=1190.127,218.481,-60.675,-177.546,6.767,148.529
C08652=1190.123,218.730,-60.699,-177.543,6.769,148.529
C08653=1190.118,218.978,-60.725,-177.541,6.771,148.528
C08654=1190.113,219.227,-60.749,-177.538,6.774,148.528
C08655=1190.108,219.475,-60.775,-177.535,6.775,148.528
C08656=1190.105,219.724,-60.799,-177.533,6.777,148.527
C08657=1190.100,219.973,-60.824,-177.530,6.779,148.527
C08658=1190.095,220.222,-60.850,-177.527,6.782,148.527
C08659=1190.091,220.470,-60.874,-177.525,6.784,148.527
C08660=1190.087,220.719,-60.900,-177.522,6.786,148.527
C08661=1190.082,220.968,-60.924,-177.520,6.788,148.526
C08662=1190.077,221.217,-60.950,-177.517,6.790,148.526
C08663=1190.072,221.465,-60.975,-177.514,6.793,148.526
C08664=1190.069,221.714,-61.000,-177.512,6.794,148.525
C08665=1190.064,221.963,-61.024,-177.509,6.796,148.525
C08666=1190.059,222.211,-61.050,-177.506,6.799,148.525
C08667=1190.054,222.460,-61.075,-177.504,6.801,148.525
C08668=1190.050,222.709,-61.101,-177.501,6.803,148.524
C08669=1190.046,222.957,-61.126,-177.498,6.806,148.524
C08670=1190.041,223.206,-61.150,-177.496,6.808,148.524
C08671=1190.037,223.455,-61.176,-177.493,6.809,148.524
C08672=1190.032,223.704,-61.201,-177.491,6.812,148.524
C08673=1190.028,223.952,-61.227,-177.488,6.814,148.523
C08674=1190.023,224.201,-61.252,-177.485,6.816,148.523
C08675=1190.018,224.450,-61.277,-177.483,6.818,148.523
C08676=1190.014,224.698,-61.302,-177.480,6.820,148.523
C08677=1190.010,224.947,-61.328,-177.477,6.823,148.522
C08678=1190.006,225.196,-61.353,-177.475,6.825,148.522
C08679=1190.001,225.444,-61.378,-177.472,6.827,148.522
C08680=1189.997,225.693,-61.404,-177.469,6.830,148.522
C08681=1189.991,225.942,-61.428,-177.467,6.831,148.521
C08682=1189.987,226.190,-61.454,-177.464,6.833,148.521
C08683=1189.982,226.438,-61.480,-177.462,6.835,148.521
C08684=1189.978,226.687,-61.505,-177.459,6.838,148.521
C08685=1189.974,226.937,-61.530,-177.457,6.840,148.521
C08686=1189.969,227.185,-61.556,-177.454,6.842,148.520
C08687=1189.965,227.434,-61.581,-177.451,6.845,148.520
C08688=1189.960,227.682,-61.607,-177.449,6.847,148.520
C08689=1189.955,227.931,-61.633,-177.446,6.849,148.519
C08690=1189.951,228.180,-61.658,-177.443,6.852,148.519
C08691=1189.946,228.428,-61.683,-177.441,6.853,148.519
C08692=1189.942,228.677,-61.709,-177.438,6.855,148.519
C08693=1189.938,228.926,-61.735,-177.436,6.857,148.519
C08694=1189.933,229.174,-61.760,-177.432,6.860,148.518
C08695=1189.929,229.423,-61.786,-177.430,6.862,148.518
C08696=1189.924,229.671,-61.811,-177.428,6.864,148.518
C08697=1189.919,229.920,-61.836,-177.424,6.867,148.518
C08698=1189.915,230.169,-61.862,-177.422,6.869,148.518
C08699=1189.911,230.418,-61.888,-177.420,6.871,148.517
C08700=1189.906,230.666,-61.913,-177.417,6.874,148.517
C08701=1189.902,230.915,-61.939,-177.414,6.875,148.517
C08702=1189.898,231.163,-61.964,-177.412,6.877,148.516
C08703=1189.893,231.412,-61.990,-177.409,6.880,148.516
C08704=1189.889,231.660,-62.016,-177.406,6.882,148.516
C08705=1189.884,231.909,-62.042,-177.404,6.884,148.516
C08706=1189.879,232.158,-62.068,-177.401,6.887,148.516
C08707=1189.874,232.406,-62.093,-177.399,6.889,148.516
C08708=1189.870,232.655,-62.119,-177.396,6.891,148.515
C08709=1189.866,232.904,-62.145,-177.393,6.893,148.515
C08710=1189.862,233.153,-62.170,-177.391,6.896,148.515
C08711=1189.857,233.401,-62.196,-177.388,6.897,148.515
C08712=1189.852,233.650,-62.222,-177.385,6.900,148.514
C08713=1189.848,233.898,-62.249,-177.383,6.902,148.514
C08714=1189.844,234.147,-62.274,-177.380,6.904,148.514
C08715=1189.839,234.395,-62.300,-177.377,6.907,148.514
C08716=1189.835,234.644,-62.325,-177.375,6.909,148.514
C08717=1189.830,234.893,-62.352,-177.372,6.911,148.513
C08718=1189.826,235.142,-62.378,-177.370,6.914,148.513
C08719=1189.821,235.390,-62.403,-177.367,6.916,148.513
C08720=1189.817,235.638,-62.429,-177.364,6.918,148.513
C08721=1189.813,235.887,-62.455,-177.362,6.921,148.513
C08722=1189.808,236.136,-62.481,-177.359,6.922,148.512
C08723=1189.802,236.407,-62.509,-177.356,6.925,148.512
C08724=1189.798,236.679,-62.538,-177.354,6.927,148.512
C08725=1189.793,236.950,-62.566,-177.350,6.930,148.512
C08726=1189.788,237.222,-62.595,-177.348,6.933,148.511
C08727=1189.783,237.470,-62.621,-177.345,6.935,148.511
C08728=1189.779,237.719,-62.646,-177.343,6.937,148.511
C08729=1189.775,237.967,-62.673,-177.340,6.940,148.511
C08730=1189.770,238.216,-62.699,-177.338,6.942,148.511
C08731=1189.766,238.465,-62.725,-177.334,6.944,148.510
C08732=1189.762,238.714,-62.751,-177.332,6.947,148.510
C08733=1189.757,238.962,-62.777,-177.330,6.948,148.510
C08734=1189.752,239.210,-62.803,-177.327,6.951,148.510
C08735=1189.748,239.459,-62.829,-177.324,6.953,148.510
C08736=1189.743,239.708,-62.856,-177.322,6.955,148.509
C08737=1189.739,239.957,-62.882,-177.319,6.958,148.509
C08738=1189.735,240.205,-62.909,-177.317,6.960,148.509
C08739=1189.730,240.454,-62.935,-177.313,6.963,148.509
C08740=1189.726,240.703,-62.960,-177.311,6.965,148.509
C08741=1189.721,240.950,-62.987,-177.309,6.967,148.508
C08742=1189.717,241.199,-63.013,-177.306,6.970,148.508
C08743=1189.712,241.448,-63.040,-177.303,6.972,148.508
C08744=1189.708,241.697,-63.066,-177.301,6.975,148.508
C08745=1189.704,241.945,-63.092,-177.298,6.976,148.508
C08746=1189.699,242.194,-63.118,-177.296,6.979,148.508
C08747=1189.695,242.442,-63.145,-177.293,6.981,148.507
C08748=1189.690,242.691,-63.171,-177.290,6.983,148.507
C08749=1189.686,242.939,-63.198,-177.288,6.986,148.507
C08750=1189.681,243.188,-63.224,-177.285,6.988,148.507
C08751=1189.677,243.436,-63.250,-177.283,6.990,148.507
C08752=1189.672,243.685,-63.276,-177.280,6.993,148.506
C08753=1189.668,243.933,-63.303,-177.277,6.995,148.506
C08754=1189.663,244.182,-63.330,-177.274,6.998,148.506
C08755=1189.659,244.431,-63.356,-177.272,7.000,148.506
C08756=1189.654,244.679,-63.383,-177.269,7.002,148.506
C08757=1189.650,244.928,-63.409,-177.267,7.005,148.506
C08758=1189.645,245.176,-63.436,-177.265,7.007,148.505
C08759=1189.641,245.424,-63.462,-177.261,7.010,148.505
C08760=1189.636,245.674,-63.488,-177.259,7.012,148.505
C08761=1189.633,245.922,-63.515,-177.257,7.014,148.505
C08762=1189.628,246.170,-63.542,-177.254,7.017,148.505
C08763=1189.624,246.419,-63.568,-177.251,7.018,148.504
C08764=1189.619,246.668,-63.595,-177.248,7.021,148.504
C08765=1189.614,246.916,-63.622,-177.246,7.024,148.504
C08766=1189.610,247.164,-63.648,-177.243,7.026,148.504
C08767=1189.605,247.413,-63.675,-177.241,7.028,148.504
C08768=1189.602,247.662,-63.701,-177.238,7.030,148.503
C08769=1189.597,247.910,-63.728,-177.236,7.033,148.503
C08770=1189.592,248.159,-63.755,-177.233,7.035,148.503
C08771=1189.588,248.407,-63.781,-177.230,7.038,148.503
C08772=1189.583,248.656,-63.808,-177.228,7.040,148.503
C08773=1189.579,248.904,-63.835,-177.225,7.043,148.503
C08774=1189.575,249.153,-63.862,-177.223,7.045,148.503
C08775=1189.570,249.401,-63.889,-177.219,7.048,148.502
C08776=1189.565,249.650,-63.916,-177.217,7.050,148.502
C08777=1189.561,249.898,-63.941,-177.215,7.052,148.502
C08778=1189.557,250.147,-63.968,-177.212,7.055,148.502
C08779=1189.552,250.396,-63.996,-177.210,7.057,148.502
C08780=1189.549,250.644,-64.022,-177.207,7.060,148.502
C08781=1189.544,250.893,-64.049,-177.204,7.062,148.501
C08782=1189.539,251.141,-64.077,-177.202,7.065,148.501
C08783=1189.535,251.390,-64.104,-177.199,7.066,148.501
C08784=1189.531,251.638,-64.130,-177.196,7.069,148.501
C08785=1189.526,251.886,-64.157,-177.194,7.072,148.501
C08786=1189.521,252.135,-64.184,-177.191,7.074,148.501
C08787=1189.517,252.383,-64.211,-177.189,7.076,148.501
C08788=1189.513,252.632,-64.238,-177.186,7.079,148.500
C08789=1189.508,252.880,-64.265,-177.183,7.081,148.500
C08790=1189.504,253.129,-64.292,-177.181,7.083,148.500
C08791=1189.499,253.378,-64.319,-177.178,7.086,148.500
C08792=1189.495,253.626,-64.346,-177.176,7.088,148.500
C08793=1189.491,253.874,-64.373,-177.173,7.091,148.500
C08794=1189.486,254.123,-64.400,-177.171,7.093,148.499
C08795=1189.482,254.371,-64.427,-177.168,7.096,148.499
C08796=1189.477,254.620,-64.454,-177.166,7.098,148.499
C08797=1189.473,254.869,-64.481,-177.162,7.101,148.499
C08798=1189.468,255.118,-64.508,-177.160,7.103,148.499
C08799=1189.464,255.366,-64.535,-177.158,7.106,148.499
C08800=1189.460,255.614,-64.563,-177.155,7.108,148.498
C08801=1189.455,255.862,-64.590,-177.152,7.111,148.498
C08802=1189.451,256.111,-64.617,-177.150,7.113,148.498
C08803=1189.447,256.360,-64.644,-177.147,7.116,148.498
C08804=1189.442,256.608,-64.671,-177.145,7.118,148.498
C08805=1189.438,256.856,-64.699,-177.142,7.121,148.498
C08806=1189.433,257.105,-64.726,-177.139,7.123,148.498
C08807=1189.428,257.353,-64.753,-177.137,7.126,148.498
C08808=1189.425,257.602,-64.780,-177.134,7.128,148.497
C08809=1189.420,257.851,-64.807,-177.131,7.130,148.497
C08810=1189.416,258.098,-64.835,-177.129,7.133,148.497
C08811=1189.411,258.347,-64.862,-177.126,7.136,148.497
C08812=1189.407,258.595,-64.889,-177.124,7.138,148.497
C08813=1189.403,258.844,-64.917,-177.121,7.140,148.497
C08814=1189.398,259.093,-64.944,-177.119,7.143,148.497
C08815=1189.394,259.341,-64.971,-177.116,7.146,148.497
C08816=1189.389,259.589,-64.999,-177.114,7.147,148.496
C08817=1189.385,259.838,-65.026,-177.111,7.150,148.496
C08818=1189.380,260.087,-65.054,-177.109,7.153,148.496
C08819=1189.376,260.334,-65.081,-177.106,7.156,148.496
C08820=1189.371,260.583,-65.108,-177.103,7.158,148.496
C08821=1189.367,260.832,-65.136,-177.101,7.160,148.496
C08822=1189.363,261.080,-65.164,-177.098,7.163,148.496
C08823=1189.358,261.329,-65.191,-177.095,7.165,148.495
C08824=1189.355,261.577,-65.219,-177.092,7.168,148.495
C08825=1189.349,261.826,-65.246,-177.090,7.170,148.495
C08826=1189.345,262.074,-65.274,-177.088,7.173,148.495
C08827=1189.341,262.347,-65.304,-177.084,7.176,148.495
C08828=1189.336,262.619,-65.335,-177.082,7.178,148.495
C08829=1189.331,262.893,-65.365,-177.079,7.181,148.495
C08830=1189.326,263.165,-65.396,-177.076,7.184,148.494
C08831=1189.321,263.414,-65.423,-177.074,7.187,148.494
C08832=1189.317,263.662,-65.451,-177.071,7.189,148.494
C08833=1189.313,263.911,-65.478,-177.068,7.192,148.494
C08834=1189.308,264.159,-65.506,-177.066,7.194,148.494
C08835=1189.304,264.408,-65.533,-177.063,7.197,148.494
C08836=1189.300,264.656,-65.561,-177.060,7.199,148.494
C08837=1189.295,264.905,-65.588,-177.058,7.202,148.494
C08838=1189.291,265.153,-65.617,-177.055,7.205,148.494
C08839=1189.286,265.401,-65.644,-177.053,7.207,148.493
C08840=1189.282,265.650,-65.671,-177.050,7.210,148.493
C08841=1189.278,265.898,-65.700,-177.048,7.212,148.493
C08842=1189.273,266.146,-65.728,-177.045,7.215,148.493
C08843=1189.269,266.396,-65.755,-177.042,7.218,148.493
C08844=1189.265,266.643,-65.783,-177.040,7.220,148.493
C08845=1189.260,266.891,-65.811,-177.037,7.222,148.493
C08846=1189.255,267.141,-65.839,-177.035,7.225,148.493
C08847=1189.251,267.389,-65.867,-177.032,7.228,148.493
C08848=1189.247,267.637,-65.895,-177.030,7.230,148.492
C08849=1189.243,267.885,-65.923,-177.027,7.233,148.492
C08850=1189.238,268.134,-65.950,-177.024,7.235,148.492
C08851=1189.234,268.383,-65.978,-177.022,7.238,148.492
C08852=1189.229,268.630,-66.006,-177.019,7.241,148.492
C08853=1189.226,268.879,-66.034,-177.017,7.243,148.492
C08854=1189.221,269.127,-66.063,-177.014,7.245,148.492
C08855=1189.216,269.376,-66.090,-177.012,7.248,148.492
C08856=1189.212,269.624,-66.118,-177.009,7.251,148.492
C08857=1189.207,269.872,-66.146,-177.006,7.254,148.492
C08858=1189.203,270.121,-66.174,-177.004,7.256,148.491
C08859=1189.199,270.369,-66.202,-177.001,7.258,148.491
C08860=1189.195,270.618,-66.231,-176.999,7.261,148.491
C08861=1189.190,270.866,-66.259,-176.996,7.264,148.491
C08862=1189.186,271.115,-66.288,-176.993,7.267,148.491
C08863=1189.181,271.363,-66.315,-176.991,7.269,148.491
C08864=1189.177,271.612,-66.343,-176.988,7.272,148.491
C08865=1189.172,271.860,-66.371,-176.986,7.274,148.491
C08866=1189.168,272.108,-66.399,-176.983,7.277,148.491
C08867=1189.163,272.357,-66.428,-176.980,7.280,148.490
C08868=1189.160,272.605,-66.456,-176.978,7.282,148.490
C08869=1189.155,272.853,-66.484,-176.975,7.285,148.490
C08870=1189.151,273.102,-66.512,-176.973,7.287,148.490
C08871=1189.146,273.350,-66.540,-176.970,7.290,148.490
C08872=1189.142,273.599,-66.569,-176.967,7.293,148.490
C08873=1189.138,273.847,-66.597,-176.965,7.295,148.490
C08874=1189.133,274.095,-66.625,-176.963,7.298,148.490
C08875=1189.129,274.343,-66.654,-176.960,7.301,148.490
C08876=1189.125,274.592,-66.683,-176.958,7.303,148.490
C08877=1189.120,274.839,-66.710,-176.954,7.306,148.489
C08878=1189.116,275.088,-66.739,-176.952,7.308,148.489
C08879=1189.112,275.337,-66.767,-176.950,7.311,148.489
C08880=1189.107,275.585,-66.796,-176.947,7.314,148.489
C08881=1189.103,275.834,-66.824,-176.945,7.316,148.489
C08882=1189.098,276.082,-66.852,-176.942,7.319,148.489
C08883=1189.095,276.330,-66.881,-176.939,7.322,148.489
C08884=1189.090,276.578,-66.909,-176.937,7.324,148.489
C08885=1189.086,276.827,-66.937,-176.934,7.327,148.489
C08886=1189.081,277.076,-66.966,-176.931,7.330,148.489
C08887=1189.077,277.323,-66.994,-176.929,7.332,148.489
C08888=1189.073,277.572,-67.023,-176.926,7.335,148.489
C08889=1189.068,277.820,-67.052,-176.924,7.337,148.489
C08890=1189.064,278.068,-67.080,-176.921,7.340,148.489
C08891=1189.060,278.317,-67.109,-176.919,7.343,148.489
C08892=1189.055,278.565,-67.137,-176.917,7.345,148.488
C08893=1189.051,278.813,-67.166,-176.913,7.348,148.488
C08894=1189.046,279.062,-67.195,-176.911,7.351,148.488
C08895=1189.042,279.310,-67.223,-176.909,7.353,148.488
C08896=1189.038,279.558,-67.252,-176.906,7.356,148.488
C08897=1189.034,279.807,-67.280,-176.903,7.359,148.488
C08898=1189.029,280.055,-67.309,-176.901,7.361,148.488
C08899=1189.025,280.304,-67.338,-176.898,7.364,148.488
C08900=1189.021,280.551,-67.367,-176.896,7.367,148.488
C08901=1189.016,280.800,-67.395,-176.893,7.369,148.488
C08902=1189.012,281.049,-67.424,-176.891,7.372,148.488
C08903=1189.008,281.297,-67.453,-176.887,7.375,148.488
C08904=1189.003,281.545,-67.481,-176.885,7.377,148.487
C08905=1188.999,281.793,-67.510,-176.883,7.380,148.487
C08906=1188.995,282.042,-67.539,-176.880,7.383,148.487
C08907=1188.991,282.289,-67.568,-176.878,7.385,148.487
C08908=1188.986,282.538,-67.596,-176.875,7.388,148.487
C08909=1188.982,282.786,-67.626,-176.872,7.391,148.487
C08910=1188.977,283.034,-67.654,-176.870,7.393,148.487
C08911=1188.973,283.283,-67.684,-176.867,7.396,148.487
C08912=1188.969,283.531,-67.712,-176.865,7.399,148.487
C08913=1188.965,283.780,-67.741,-176.863,7.402,148.487
C08914=1188.960,284.028,-67.770,-176.860,7.405,148.487
C08915=1188.955,284.276,-67.799,-176.857,7.408,148.487
C08916=1188.951,284.525,-67.828,-176.855,7.410,148.487
C08917=1188.948,284.773,-67.857,-176.852,7.413,148.487
C08918=1188.943,285.020,-67.886,-176.849,7.416,148.487
C08919=1188.938,285.269,-67.915,-176.847,7.418,148.487
C08920=1188.934,285.518,-67.944,-176.844,7.421,148.486
C08921=1188.930,285.766,-67.973,-176.841,7.424,148.486
C08922=1188.925,286.014,-68.002,-176.839,7.427,148.486
C08923=1188.921,286.262,-68.031,-176.837,7.429,148.486
C08924=1188.917,286.510,-68.060,-176.834,7.432,148.486
C08925=1188.913,286.759,-68.089,-176.831,7.435,148.486
C08926=1188.908,287.007,-68.118,-176.829,7.437,148.486
C08927=1188.904,287.255,-68.147,-176.826,7.440,148.486
C08928=1188.900,287.503,-68.177,-176.824,7.443,148.486
C08929=1188.895,287.752,-68.206,-176.821,7.445,148.486
C08930=1188.891,288.000,-68.235,-176.819,7.448,148.486
C08931=1188.886,288.275,-68.267,-176.816,7.451,148.486
C08932=1188.881,288.549,-68.300,-176.813,7.454,148.486
C08933=1188.877,288.824,-68.332,-176.811,7.457,148.486
C08934=1188.872,289.098,-68.364,-176.807,7.461,148.486
C08935=1188.868,289.347,-68.393,-176.805,7.463,148.486
C08936=1188.863,289.595,-68.422,-176.802,7.466,148.486
C08937=1188.859,289.843,-68.452,-176.800,7.469,148.486
C08938=1188.855,290.091,-68.481,-176.798,7.471,148.486
C08939=1188.851,290.340,-68.511,-176.795,7.474,148.486
C08940=1188.846,290.587,-68.540,-176.792,7.477,148.486
C08941=1188.842,290.835,-68.569,-176.789,7.480,148.486
C08942=1188.838,291.084,-68.599,-176.787,7.483,148.486
C08943=1188.834,291.332,-68.628,-176.785,7.486,148.486
C08944=1188.829,291.580,-68.657,-176.782,7.489,148.486
C08945=1188.824,291.829,-68.688,-176.780,7.491,148.486
C08946=1188.820,292.077,-68.717,-176.777,7.494,148.485
C08947=1188.816,292.326,-68.746,-176.774,7.497,148.485
C08948=1188.812,292.574,-68.775,-176.772,7.500,148.485
C08949=1188.807,292.821,-68.805,-176.769,7.502,148.485
C08950=1188.803,293.069,-68.834,-176.767,7.505,148.485
C08951=1188.799,293.318,-68.864,-176.764,7.508,148.485
C08952=1188.795,293.566,-68.893,-176.761,7.511,148.485
C08953=1188.790,293.814,-68.923,-176.759,7.513,148.485
C08954=1188.786,294.062,-68.952,-176.756,7.516,148.485
C08955=1188.782,294.311,-68.982,-176.754,7.519,148.485
C08956=1188.777,294.559,-69.012,-176.751,7.522,148.485
C08957=1188.773,294.808,-69.041,-176.749,7.524,148.485
C08958=1188.769,295.056,-69.071,-176.746,7.527,148.485
C08959=1188.765,295.304,-69.100,-176.743,7.530,148.485
C08960=1188.761,295.552,-69.130,-176.741,7.533,148.485
C08961=1188.757,295.800,-69.160,-176.739,7.535,148.485
C08962=1188.752,296.049,-69.190,-176.736,7.539,148.485
C08963=1188.747,296.297,-69.219,-176.734,7.542,148.485
C08964=1188.743,296.545,-69.249,-176.731,7.545,148.485
C08965=1188.739,296.793,-69.279,-176.729,7.547,148.485
C08966=1188.735,297.041,-69.308,-176.726,7.550,148.485
C08967=1188.730,297.290,-69.338,-176.723,7.553,148.485
C08968=1188.726,297.538,-69.368,-176.721,7.556,148.485
C08969=1188.722,297.786,-69.398,-176.718,7.558,148.485
C08970=1188.718,298.034,-69.427,-176.716,7.561,148.485
C08971=1188.713,298.282,-69.457,-176.713,7.564,148.485
C08972=1188.709,298.531,-69.487,-176.710,7.567,148.485
C08973=1188.705,298.778,-69.517,-176.709,7.570,148.485
C08974=1188.701,299.027,-69.547,-176.706,7.573,148.485
C08975=1188.696,299.275,-69.577,-176.703,7.576,148.485
C08976=1188.692,299.523,-69.607,-176.700,7.579,148.485
C08977=1188.688,299.771,-69.636,-176.698,7.581,148.485
C08978=1188.683,300.019,-69.667,-176.696,7.584,148.485
C08979=1188.679,300.267,-69.696,-176.693,7.587,148.485
C08980=1188.675,300.516,-69.726,-176.690,7.590,148.485
C08981=1188.670,300.764,-69.757,-176.688,7.592,148.485
C08982=1188.666,301.012,-69.786,-176.686,7.595,148.485
C08983=1188.662,301.259,-69.816,-176.683,7.598,148.485
C08984=1188.657,301.508,-69.846,-176.680,7.601,148.485
C08985=1188.654,301.756,-69.877,-176.678,7.604,148.485
C08986=1188.649,302.005,-69.907,-176.676,7.606,148.485
C08987=1188.645,302.253,-69.937,-176.673,7.609,148.485
C08988=1188.641,302.501,-69.967,-176.670,7.612,148.485
C08989=1188.636,302.749,-69.997,-176.667,7.615,148.485
C08990=1188.632,302.997,-70.027,-176.666,7.618,148.485
C08991=1188.628,303.245,-70.058,-176.663,7.621,148.485
C08992=1188.624,303.493,-70.087,-176.660,7.624,148.485
C08993=1188.619,303.741,-70.118,-176.658,7.627,148.485
C08994=1188.615,303.990,-70.148,-176.655,7.630,148.485
C08995=1188.611,304.238,-70.178,-176.653,7.632,148.485
C08996=1188.607,304.486,-70.209,-176.650,7.635,148.485
C08997=1188.603,304.734,-70.238,-176.648,7.638,148.485
C08998=1188.598,304.982,-70.269,-176.645,7.641,148.485
C08999=1188.593,305.230,-70.299,-176.642,7.644,148.485
C09000=1188.589,305.478,-70.329,-176.640,7.647,148.485
C09001=1188.585,305.727,-70.360,-176.638,7.650,148.485
C09002=1188.581,305.975,-70.390,-176.635,7.653,148.485
C09003=1188.576,306.223,-70.420,-176.632,7.656,148.485
C09004=1188.573,306.471,-70.450,-176.630,7.659,148.485
C09005=1188.568,306.719,-70.481,-176.628,7.661,148.485
C09006=1188.564,306.966,-70.511,-176.625,7.664,148.485
C09007=1188.560,307.216,-70.542,-176.623,7.667,148.485
C09008=1188.556,307.463,-70.572,-176.620,7.670,148.485
C09009=1188.551,307.711,-70.603,-176.617,7.673,148.485
C09010=1188.547,307.959,-70.633,-176.615,7.676,148.485
C09011=1188.542,308.208,-70.663,-176.613,7.679,148.485
C09012=1188.538,308.456,-70.694,-176.610,7.682,148.485
C09013=1188.535,308.704,-70.724,-176.607,7.685,148.485
C09014=1188.530,308.952,-70.755,-176.605,7.688,148.485
C09015=1188.525,309.200,-70.786,-176.603,7.690,148.485
C09016=1188.522,309.448,-70.816,-176.600,7.693,148.485
C09017=1188.517,309.696,-70.847,-176.598,7.696,148.485
C09018=1188.513,309.945,-70.877,-176.595,7.699,148.485
C09019=1188.509,310.192,-70.907,-176.592,7.702,148.485
C09020=1188.505,310.441,-70.938,-176.591,7.705,148.485
C09021=1188.500,310.689,-70.969,-176.588,7.708,148.485
C09022=1188.496,310.937,-70.999,-176.585,7.711,148.485
C09023=1188.492,311.185,-71.030,-176.582,7.714,148.485
C09024=1188.488,311.433,-71.061,-176.580,7.717,148.486
C09025=1188.484,311.681,-71.091,-176.577,7.720,148.486
C09026=1188.479,311.929,-71.122,-176.575,7.723,148.485
C09027=1188.475,312.177,-71.153,-176.573,7.726,148.485
C09028=1188.470,312.425,-71.184,-176.570,7.729,148.486
C09029=1188.467,312.673,-71.214,-176.568,7.732,148.486
C09030=1188.462,312.921,-71.245,-176.565,7.735,148.486
C09031=1188.458,313.170,-71.276,-176.563,7.738,148.486
C09032=1188.453,313.418,-71.307,-176.561,7.740,148.486
C09033=1188.449,313.665,-71.337,-176.558,7.743,148.486
C09034=1188.446,313.913,-71.369,-176.555,7.746,148.486
C09035=1188.441,314.190,-71.402,-176.553,7.750,148.486
C09036=1188.436,314.467,-71.438,-176.550,7.754,148.486
C09037=1188.432,314.743,-71.472,-176.547,7.757,148.486
C09038=1188.426,315.019,-71.506,-176.544,7.760,148.486
C09039=1188.422,315.268,-71.537,-176.542,7.763,148.486
C09040=1188.418,315.515,-71.569,-176.539,7.766,148.486
C09041=1188.414,315.763,-71.599,-176.537,7.769,148.486
C09042=1188.410,316.012,-71.630,-176.535,7.771,148.486
C09043=1188.406,316.260,-71.661,-176.532,7.774,148.486
C09044=1188.401,316.507,-71.692,-176.529,7.777,148.486
C09045=1188.397,316.756,-71.723,-176.527,7.781,148.487
C09046=1188.393,317.004,-71.754,-176.524,7.784,148.486
C09047=1188.389,317.252,-71.785,-176.522,7.787,148.486
C09048=1188.384,317.500,-71.817,-176.520,7.789,148.487
C09049=1188.380,317.748,-71.847,-176.517,7.792,148.487
C09050=1188.376,317.996,-71.878,-176.515,7.795,148.487
C09051=1188.371,318.244,-71.910,-176.512,7.799,148.487
C09052=1188.367,318.492,-71.941,-176.510,7.802,148.487
C09053=1188.364,318.740,-71.971,-176.507,7.805,148.487
C09054=1188.360,318.988,-72.003,-176.505,7.808,148.487
C09055=1188.355,319.236,-72.034,-176.503,7.810,148.487
C09056=1188.351,319.484,-72.065,-176.500,7.813,148.487
C09057=1188.347,319.732,-72.096,-176.498,7.816,148.487
C09058=1188.342,319.980,-72.127,-176.495,7.819,148.487
C09059=1188.339,320.228,-72.159,-176.493,7.823,148.487
C09060=1188.334,320.476,-72.190,-176.490,7.826,148.487
C09061=1188.330,320.724,-72.222,-176.488,7.828,148.488
C09062=1188.326,320.972,-72.252,-176.486,7.831,148.488
C09063=1188.322,321.220,-72.284,-176.483,7.835,148.488
C09064=1188.317,321.468,-72.315,-176.481,7.838,148.488
C09065=1188.314,321.716,-72.347,-176.478,7.841,148.488
C09066=1188.309,321.964,-72.378,-176.476,7.844,148.488
C09067=1188.305,322.212,-72.410,-176.473,7.847,148.488
C09068=1188.301,322.460,-72.440,-176.471,7.849,148.488
C09069=1188.296,322.708,-72.473,-176.469,7.852,148.488
C09070=1188.292,322.956,-72.503,-176.466,7.856,148.488
C09071=1188.288,323.204,-72.535,-176.464,7.859,148.488
C09072=1188.284,323.452,-72.567,-176.461,7.862,148.488
C09073=1188.280,323.700,-72.598,-176.459,7.865,148.488
C09074=1188.275,323.948,-72.629,-176.456,7.868,148.488
C09075=1188.271,324.196,-72.661,-176.454,7.871,148.489
C09076=1188.267,324.444,-72.692,-176.452,7.874,148.489
C09077=1188.263,324.692,-72.724,-176.449,7.877,148.489
C09078=1188.259,324.940,-72.755,-176.447,7.880,148.489
C09079=1188.254,325.188,-72.787,-176.444,7.883,148.489
C09080=1188.251,325.436,-72.819,-176.442,7.886,148.489
C09081=1188.246,325.683,-72.850,-176.439,7.890,148.489
C09082=1188.242,325.932,-72.882,-176.437,7.893,148.489
C09083=1188.238,326.179,-72.913,-176.435,7.895,148.489
C09084=1188.233,326.428,-72.945,-176.432,7.898,148.489
C09085=1188.230,326.676,-72.977,-176.430,7.901,148.490
C09086=1188.225,326.924,-73.008,-176.427,7.904,148.490
C09087=1188.221,327.172,-73.040,-176.425,7.908,148.490
C09088=1188.217,327.419,-73.071,-176.422,7.911,148.490
C09089=1188.213,327.667,-73.104,-176.420,7.914,148.490
C09090=1188.209,327.915,-73.136,-176.417,7.917,148.490
C09091=1188.204,328.163,-73.166,-176.416,7.920,148.490
C09092=1188.201,328.411,-73.198,-176.414,7.923,148.490
C09093=1188.196,328.659,-73.230,-176.411,7.926,148.490
C09094=1188.192,328.907,-73.262,-176.409,7.929,148.491
C09095=1188.188,329.155,-73.294,-176.406,7.932,148.491
C09096=1188.183,329.403,-73.326,-176.404,7.936,148.491
C09097=1188.179,329.651,-73.358,-176.401,7.939,148.491
C09098=1188.176,329.899,-73.390,-176.399,7.942,148.491
C09099=1188.171,330.146,-73.421,-176.397,7.944,148.491
C09100=1188.167,330.395,-73.454,-176.394,7.947,148.491
C09101=1188.163,330.643,-73.486,-176.392,7.951,148.491
C09102=1188.159,330.890,-73.517,-176.389,7.954,148.491
C09103=1188.155,331.138,-73.549,-176.387,7.957,148.492
C09104=1188.151,331.386,-73.581,-176.385,7.960,148.492
C09105=1188.146,331.634,-73.613,-176.382,7.963,148.492
C09106=1188.142,331.882,-73.645,-176.380,7.967,148.492
C09107=1188.138,332.130,-73.677,-176.378,7.970,148.492
C09108=1188.133,332.378,-73.709,-176.375,7.972,148.492
C09109=1188.130,332.626,-73.741,-176.373,7.975,148.492
C09110=1188.125,332.874,-73.773,-176.371,7.978,148.492
C09111=1188.121,333.121,-73.805,-176.368,7.982,148.493
C09112=1188.117,333.369,-73.837,-176.366,7.985,148.493
C09113=1188.113,333.618,-73.869,-176.363,7.988,148.493
C09114=1188.109,333.866,-73.901,-176.361,7.991,148.493
C09115=1188.104,334.113,-73.934,-176.359,7.995,148.493
C09116=1188.101,334.361,-73.966,-176.356,7.998,148.493
C09117=1188.096,334.609,-73.998,-176.354,8.000,148.493
C09118=1188.092,334.857,-74.030,-176.352,8.004,148.494
C09119=1188.087,335.105,-74.062,-176.350,8.007,148.494
C09120=1188.084,335.352,-74.095,-176.347,8.010,148.494
C09121=1188.080,335.601,-74.127,-176.345,8.013,148.494
C09122=1188.076,335.849,-74.159,-176.343,8.017,148.494
C09123=1188.071,336.096,-74.191,-176.340,8.020,148.494
C09124=1188.067,336.344,-74.224,-176.338,8.023,148.495
C09125=1188.063,336.592,-74.256,-176.336,8.026,148.495
C09126=1188.059,336.840,-74.288,-176.334,8.029,148.495
C09127=1188.055,337.089,-74.320,-176.331,8.032,148.495
C09128=1188.051,337.335,-74.352,-176.329,8.035,148.495
C09129=1188.046,337.584,-74.385,-176.327,8.038,148.495
C09130=1188.043,337.832,-74.417,-176.324,8.042,148.496
C09131=1188.038,338.079,-74.450,-176.322,8.045,148.496
C09132=1188.034,338.328,-74.482,-176.319,8.048,148.496
C09133=1188.030,338.574,-74.515,-176.317,8.051,148.496
C09134=1188.026,338.823,-74.547,-176.315,8.055,148.496
C09135=1188.022,339.071,-74.579,-176.313,8.058,148.496
C09136=1188.018,339.319,-74.612,-176.311,8.060,148.496
C09137=1188.013,339.567,-74.644,-176.308,8.064,148.497
C09138=1188.010,339.814,-74.677,-176.306,8.067,148.497
